gfCNCPoint3[16834] = {X 95.6267, Y 61.5566, Z -4.6667, A 0.000, B 0.000, C 0.000 }
gfCNCPoint3[16835] = {X 93.9906, Y 61.7990, Z -4.6667, A 0.000, B 0.000, C 0.000 }
gfCNCPoint3[16836] = {X 92.3385, Y 61.8800, Z -4.6667, A 0.000, B 0.000, C 0.000 }
gfCNCPoint3[16837] = {X 85.8951, Y 61.8800, Z -4.6667, A 0.000, B 0.000, C 0.000 }
gfCNCPoint3[16838] = {X 85.1609, Y 61.8640, Z -4.6667, A 0.000, B 0.000, C 0.000 }
gfCNCPoint3[16839] = {X 84.4280, Y 61.8161, Z -4.6667, A 0.000, B 0.000, C 0.000 }
gfCNCPoint3[16840] = {X 82.7247, Y 63.0692, Z -4.6667, A 0.000, B 0.000, C 0.000 }
gfCNCPoint3[16841] = {X 80.9073, Y 64.1504, Z -4.6667, A 0.000, B 0.000, C 0.000 }
gfCNCPoint3[16842] = {X 78.9932, Y 65.0494, Z -4.6667, A 0.000, B 0.000, C 0.000 }
gfCNCPoint3[16843] = {X 77.0007, Y 65.7577, Z -4.6667, A 0.000, B 0.000, C 0.000 }
gfCNCPoint3[16844] = {X 74.9487, Y 66.2685, Z -4.6667, A 0.000, B 0.000, C 0.000 }
gfCNCPoint3[16845] = {X 72.8566, Y 66.5769, Z -4.6667, A 0.000, B 0.000, C 0.000 }
gfCNCPoint3[16846] = {X 70.7445, Y 66.6800, Z -4.6667, A 0.000, B 0.000, C 0.000 }
gfCNCPoint3[16847] = {X 64.1851, Y 66.6800, Z -4.6667, A 0.000, B 0.000, C 0.000 }
gfCNCPoint3[16848] = {X 62.0576, Y 66.5754, Z -4.6667, A 0.000, B 0.000, C 0.000 }
gfCNCPoint3[16849] = {X 59.9505, Y 66.2624, Z -4.6667, A 0.000, B 0.000, C 0.000 }
gfCNCPoint3[16850] = {X 57.8844, Y 65.7442, Z -4.6667, A 0.000, B 0.000, C 0.000 }
gfCNCPoint3[16851] = {X 55.8790, Y 65.0258, Z -4.6667, A 0.000, B 0.000, C 0.000 }
gfCNCPoint3[16852] = {X 53.8737, Y 65.7442, Z -4.6667, A 0.000, B 0.000, C 0.000 }
gfCNCPoint3[16853] = {X 51.8075, Y 66.2624, Z -4.6667, A 0.000, B 0.000, C 0.000 }
gfCNCPoint3[16854] = {X 49.7005, Y 66.5754, Z -4.6667, A 0.000, B 0.000, C 0.000 }
gfCNCPoint3[16855] = {X 47.5729, Y 66.6800, Z -4.6667, A 0.000, B 0.000, C 0.000 }
gfCNCPoint3[16856] = {X 40.6393, Y 66.6800, Z -4.6667, A 0.000, B 0.000, C 0.000 }
gfCNCPoint3[16857] = {X 38.5447, Y 66.5786, Z -4.6667, A 0.000, B 0.000, C 0.000 }
gfCNCPoint3[16858] = {X 36.4697, Y 66.2753, Z -4.6667, A 0.000, B 0.000, C 0.000 }
gfCNCPoint3[16859] = {X 34.5048, Y 67.0013, Z -4.6667, A 0.000, B 0.000, C 0.000 }
gfCNCPoint3[16860] = {X 32.4879, Y 67.5668, Z -4.6667, A 0.000, B 0.000, C 0.000 }
gfCNCPoint3[16861] = {X 30.4319, Y 67.9682, Z -4.6667, A 0.000, B 0.000, C 0.000 }
gfCNCPoint3[16862] = {X 28.4180, Y 68.7658, Z -4.6667, A 0.000, B 0.000, C 0.000 }
gfCNCPoint3[16863] = {X 26.3720, Y 69.4768, Z -4.6667, A 0.000, B 0.000, C 0.000 }
gfCNCPoint3[16864] = {X 23.9561, Y 70.1952, Z -4.6667, A 0.000, B 0.000, C 0.000 }
gfCNCPoint3[16865] = {X 21.5034, Y 70.7756, Z -4.6667, A 0.000, B 0.000, C 0.000 }
gfCNCPoint3[16866] = {X 21.5034, Y 78.4950, Z -4.6667, A 0.000, B 0.000, C 0.000 }
gfCNCPoint3[16867] = {X 109.6713, Y 78.4950, Z -4.6667, A 0.000, B 0.000, C 0.000 }
gfCNCPoint3[16868] = {X 111.3427, Y 77.2335, Z -4.6667, A 0.000, B 0.000, C 0.000 }
gfCNCPoint3[16869] = {X 113.1173, Y 76.1220, Z -4.6667, A 0.000, B 0.000, C 0.000 }
gfCNCPoint3[16870] = {X 114.9818, Y 75.1689, Z -4.6667, A 0.000, B 0.000, C 0.000 }
gfCNCPoint3[16871] = {X 116.9220, Y 74.3813, Z -4.6667, A 0.000, B 0.000, C 0.000 }
gfCNCPoint3[16872] = {X 130.4111, Y 59.5684, Z -4.6667, A 0.000, B 0.000, C 0.000 }
gfCNCPoint3[16873] = {X 129.5278, Y 58.7531, Z -4.6667, A 0.000, B 0.000, C 0.000 }
gfCNCPoint3[16874] = {X 128.6970, Y 57.8844, Z -4.6667, A 0.000, B 0.000, C 0.000 }
gfCNCPoint3[16875] = {X 127.3929, Y 58.8834, Z -4.6667, A 0.000, B 0.000, C 0.000 }
gfCNCPoint3[16876] = {X 125.9978, Y 59.7510, Z -4.6667, A 0.000, B 0.000, C 0.000 }
gfCNCPoint3[16877] = {X 124.5250, Y 60.4789, Z -4.6667, A 0.000, B 0.000, C 0.000 }
gfCNCPoint3[16878] = {X 122.9885, Y 61.0601, Z -4.6667, A 0.000, B 0.000, C 0.000 }
gfCNCPoint3[16879] = {X 121.2879, Y 61.5139, Z -4.6667, A 0.000, B 0.000, C 0.000 }
gfCNCPoint3[16880] = {X 119.5493, Y 61.7882, Z -4.6667, A 0.000, B 0.000, C 0.000 }
gfCNCPoint3[16881] = {X 117.7916, Y 61.8800, Z -4.6667, A 0.000, B 0.000, C 0.000 }
gfCNCPoint3[16882] = {X 111.9185, Y 61.8800, Z -4.6667, A 0.000, B 0.000, C 0.000 }
gfCNCPoint3[16883] = {X 111.6170, Y 61.8773, Z -4.6667, A 0.000, B 0.000, C 0.000 }
gfCNCPoint3[16884] = {X 111.3156, Y 61.8692, Z -4.6667, A 0.000, B 0.000, C 0.000 }
gfCNCPoint3[16885] = {X 111.4013, Y 59.4708, Z -4.6667, A 0.000, B 0.000, C 0.000 }
gfCNCPoint3[16886] = {X 109.9149, Y 59.3407, Z -4.6667, A 0.000, B 0.000, C 0.000 }
gfCNCPoint3[16887] = {X 108.4496, Y 59.0584, Z -4.6667, A 0.000, B 0.000, C 0.000 }
gfCNCPoint3[16888] = {X 107.0213, Y 58.6267, Z -4.6667, A 0.000, B 0.000, C 0.000 }
gfCNCPoint3[16889] = {X 105.4260, Y 59.0985, Z -4.6667, A 0.000, B 0.000, C 0.000 }
gfCNCPoint3[16890] = {X 103.7872, Y 59.3842, Z -4.6667, A 0.000, B 0.000, C 0.000 }
gfCNCPoint3[16891] = {X 102.1264, Y 59.4800, Z -4.6667, A 0.000, B 0.000, C 0.000 }
gfCNCPoint3[16892] = {X 100.4656, Y 59.3847, Z -4.6667, A 0.000, B 0.000, C 0.000 }
gfCNCPoint3[16893] = {X 98.8267, Y 59.0996, Z -4.6667, A 0.000, B 0.000, C 0.000 }
gfCNCPoint3[16894] = {X 97.2313, Y 58.6283, Z -4.6667, A 0.000, B 0.000, C 0.000 }
gfCNCPoint3[16895] = {X 95.6367, Y 59.0994, Z -4.6667, A 0.000, B 0.000, C 0.000 }
gfCNCPoint3[16896] = {X 93.9986, Y 59.3845, Z -4.6667, A 0.000, B 0.000, C 0.000 }
gfCNCPoint3[16897] = {X 92.3385, Y 59.4800, Z -4.6667, A 0.000, B 0.000, C 0.000 }
gfCNCPoint3[16898] = {X 85.8951, Y 59.4800, Z -4.6667, A 0.000, B 0.000, C 0.000 }
gfCNCPoint3[16899] = {X 84.7780, Y 59.4368, Z -4.6667, A 0.000, B 0.000, C 0.000 }
gfCNCPoint3[16900] = {X 83.6677, Y 59.3077, Z -4.6667, A 0.000, B 0.000, C 0.000 }
gfCNCPoint3[16901] = {X 82.0978, Y 60.5827, Z -4.6667, A 0.000, B 0.000, C 0.000 }
gfCNCPoint3[16902] = {X 80.4031, Y 61.6862, Z -4.6667, A 0.000, B 0.000, C 0.000 }
gfCNCPoint3[16903] = {X 78.6021, Y 62.6061, Z -4.6667, A 0.000, B 0.000, C 0.000 }
gfCNCPoint3[16904] = {X 76.7146, Y 63.3324, Z -4.6667, A 0.000, B 0.000, C 0.000 }
gfCNCPoint3[16905] = {X 74.7614, Y 63.8569, Z -4.6667, A 0.000, B 0.000, C 0.000 }
gfCNCPoint3[16906] = {X 72.7640, Y 64.1739, Z -4.6667, A 0.000, B 0.000, C 0.000 }
gfCNCPoint3[16907] = {X 70.7445, Y 64.2800, Z -4.6667, A 0.000, B 0.000, C 0.000 }
gfCNCPoint3[16908] = {X 64.1851, Y 64.2800, Z -4.6667, A 0.000, B 0.000, C 0.000 }
gfCNCPoint3[16909] = {X 62.0428, Y 64.1606, Z -4.6667, A 0.000, B 0.000, C 0.000 }
gfCNCPoint3[16910] = {X 59.9269, Y 63.8039, Z -4.6667, A 0.000, B 0.000, C 0.000 }
gfCNCPoint3[16911] = {X 57.8638, Y 63.2143, Z -4.6667, A 0.000, B 0.000, C 0.000 }
gfCNCPoint3[16912] = {X 55.8790, Y 62.3991, Z -4.6667, A 0.000, B 0.000, C 0.000 }
gfCNCPoint3[16913] = {X 53.8942, Y 63.2143, Z -4.6667, A 0.000, B 0.000, C 0.000 }
gfCNCPoint3[16914] = {X 51.8311, Y 63.8039, Z -4.6667, A 0.000, B 0.000, C 0.000 }
gfCNCPoint3[16915] = {X 49.7153, Y 64.1606, Z -4.6667, A 0.000, B 0.000, C 0.000 }
gfCNCPoint3[16916] = {X 47.5729, Y 64.2800, Z -4.6667, A 0.000, B 0.000, C 0.000 }
gfCNCPoint3[16917] = {X 40.6393, Y 64.2800, Z -4.6667, A 0.000, B 0.000, C 0.000 }
gfCNCPoint3[16918] = {X 39.1549, Y 64.2228, Z -4.6667, A 0.000, B 0.000, C 0.000 }
gfCNCPoint3[16919] = {X 37.6792, Y 64.0514, Z -4.6667, A 0.000, B 0.000, C 0.000 }
gfCNCPoint3[16920] = {X 36.2212, Y 63.7670, Z -4.6667, A 0.000, B 0.000, C 0.000 }
gfCNCPoint3[16921] = {X 34.1358, Y 64.5944, Z -4.6667, A 0.000, B 0.000, C 0.000 }
gfCNCPoint3[16922] = {X 31.9814, Y 65.2203, Z -4.6667, A 0.000, B 0.000, C 0.000 }
gfCNCPoint3[16923] = {X 29.7773, Y 65.6388, Z -4.6667, A 0.000, B 0.000, C 0.000 }
gfCNCPoint3[16924] = {X 27.7204, Y 66.4644, Z -4.6667, A 0.000, B 0.000, C 0.000 }
gfCNCPoint3[16925] = {X 25.6278, Y 67.1951, Z -4.6667, A 0.000, B 0.000, C 0.000 }
gfCNCPoint3[16926] = {X 23.4821, Y 67.8375, Z -4.6667, A 0.000, B 0.000, C 0.000 }
gfCNCPoint3[16927] = {X 21.3053, Y 68.3647, Z -4.6667, A 0.000, B 0.000, C 0.000 }
gfCNCPoint3[16928] = {X 19.1034, Y 68.7753, Z -4.6667, A 0.000, B 0.000, C 0.000 }
gfCNCPoint3[16929] = {X 19.1034, Y 80.8950, Z -4.6667, A 0.000, B 0.000, C 0.000 }
gfCNCPoint3[16930] = {X 110.5596, Y 80.8950, Z -4.6667, A 0.000, B 0.000, C 0.000 }
gfCNCPoint3[16931] = {X 112.3069, Y 79.4902, Z -4.6667, A 0.000, B 0.000, C 0.000 }
gfCNCPoint3[16932] = {X 114.1898, Y 78.2733, Z -4.6667, A 0.000, B 0.000, C 0.000 }
gfCNCPoint3[16933] = {X 116.1884, Y 77.2574, Z -4.6667, A 0.000, B 0.000, C 0.000 }
gfCNCPoint3[16934] = {X 118.2812, Y 76.4533, Z -4.6667, A 0.000, B 0.000, C 0.000 }
gfCNCPoint3[16935] = {X 133.9633, Y 59.2322, Z -4.6667, A 0.000, B 0.000, C 0.000 }
gfCNCPoint3[16936] = {X 132.7155, Y 58.3546, Z -4.6667, A 0.000, B 0.000, C 0.000 }
gfCNCPoint3[16937] = {X 131.5520, Y 57.3681, Z -4.6667, A 0.000, B 0.000, C 0.000 }
gfCNCPoint3[16938] = {X 130.4824, Y 56.2805, Z -4.6667, A 0.000, B 0.000, C 0.000 }
gfCNCPoint3[16939] = {X 129.6655, Y 55.2988, Z -4.6667, A 0.000, B 0.000, C 0.000 }
gfCNCPoint3[16940] = {X 128.9251, Y 54.2582, Z -4.6667, A 0.000, B 0.000, C 0.000 }
gfCNCPoint3[16941] = {X 128.0750, Y 55.1942, Z -4.6667, A 0.000, B 0.000, C 0.000 }
gfCNCPoint3[16942] = {X 127.1464, Y 56.0525, Z -4.6667, A 0.000, B 0.000, C 0.000 }
gfCNCPoint3[16943] = {X 125.7915, Y 57.0695, Z -4.6667, A 0.000, B 0.000, C 0.000 }
gfCNCPoint3[16944] = {X 124.3270, Y 57.9212, Z -4.6667, A 0.000, B 0.000, C 0.000 }
gfCNCPoint3[16945] = {X 122.7731, Y 58.5961, Z -4.6667, A 0.000, B 0.000, C 0.000 }
gfCNCPoint3[16946] = {X 121.1510, Y 59.0849, Z -4.6667, A 0.000, B 0.000, C 0.000 }
gfCNCPoint3[16947] = {X 119.4828, Y 59.3809, Z -4.6667, A 0.000, B 0.000, C 0.000 }
gfCNCPoint3[16948] = {X 117.7916, Y 59.4800, Z -4.6667, A 0.000, B 0.000, C 0.000 }
gfCNCPoint3[16949] = {X 111.9185, Y 59.4800, Z -4.6667, A 0.000, B 0.000, C 0.000 }
gfCNCPoint3[16950] = {X 111.6599, Y 59.4777, Z -4.6667, A 0.000, B 0.000, C 0.000 }
gfCNCPoint3[16951] = {X 111.4013, Y 59.4708, Z -4.6667, A 0.000, B 0.000, C 0.000 }
gfCNCPoint3[16952] = {X 111.4871, Y 57.0723, Z -4.6667, A 0.000, B 0.000, C 0.000 }
gfCNCPoint3[16953] = {X 109.9587, Y 56.9200, Z -4.6667, A 0.000, B 0.000, C 0.000 }
gfCNCPoint3[16954] = {X 108.4621, Y 56.5750, Z -4.6667, A 0.000, B 0.000, C 0.000 }
gfCNCPoint3[16955] = {X 107.0213, Y 56.0428, Z -4.6667, A 0.000, B 0.000, C 0.000 }
gfCNCPoint3[16956] = {X 105.4432, Y 56.6151, Z -4.6667, A 0.000, B 0.000, C 0.000 }
gfCNCPoint3[16957] = {X 103.8010, Y 56.9630, Z -4.6667, A 0.000, B 0.000, C 0.000 }
gfCNCPoint3[16958] = {X 102.1265, Y 57.0800, Z -4.6667, A 0.000, B 0.000, C 0.000 }
gfCNCPoint3[16959] = {X 100.4519, Y 56.9637, Z -4.6667, A 0.000, B 0.000, C 0.000 }
gfCNCPoint3[16960] = {X 98.8096, Y 56.6164, Z -4.6667, A 0.000, B 0.000, C 0.000 }
gfCNCPoint3[16961] = {X 97.2313, Y 56.0448, Z -4.6667, A 0.000, B 0.000, C 0.000 }
gfCNCPoint3[16962] = {X 95.6538, Y 56.6162, Z -4.6667, A 0.000, B 0.000, C 0.000 }
gfCNCPoint3[16963] = {X 94.0123, Y 56.9635, Z -4.6667, A 0.000, B 0.000, C 0.000 }
gfCNCPoint3[16964] = {X 92.3385, Y 57.0800, Z -4.6667, A 0.000, B 0.000, C 0.000 }
gfCNCPoint3[16965] = {X 85.8951, Y 57.0800, Z -4.6667, A 0.000, B 0.000, C 0.000 }
gfCNCPoint3[16966] = {X 84.3894, Y 56.9858, Z -4.6667, A 0.000, B 0.000, C 0.000 }
gfCNCPoint3[16967] = {X 82.9073, Y 56.7047, Z -4.6667, A 0.000, B 0.000, C 0.000 }
gfCNCPoint3[16968] = {X 81.4847, Y 58.0224, Z -4.6667, A 0.000, B 0.000, C 0.000 }
gfCNCPoint3[16969] = {X 79.9203, Y 59.1682, Z -4.6667, A 0.000, B 0.000, C 0.000 }
gfCNCPoint3[16970] = {X 78.2348, Y 60.1271, Z -4.6667, A 0.000, B 0.000, C 0.000 }
gfCNCPoint3[16971] = {X 76.4504, Y 60.8864, Z -4.6667, A 0.000, B 0.000, C 0.000 }
gfCNCPoint3[16972] = {X 74.5908, Y 61.4359, Z -4.6667, A 0.000, B 0.000, C 0.000 }
gfCNCPoint3[16973] = {X 72.6804, Y 61.7686, Z -4.6667, A 0.000, B 0.000, C 0.000 }
gfCNCPoint3[16974] = {X 70.7445, Y 61.8800, Z -4.6667, A 0.000, B 0.000, C 0.000 }
gfCNCPoint3[16975] = {X 64.1851, Y 61.8800, Z -4.6667, A 0.000, B 0.000, C 0.000 }
gfCNCPoint3[16976] = {X 62.4514, Y 61.7907, Z -4.6667, A 0.000, B 0.000, C 0.000 }
gfCNCPoint3[16977] = {X 60.7359, Y 61.5238, Z -4.6667, A 0.000, B 0.000, C 0.000 }
gfCNCPoint3[16978] = {X 59.0570, Y 61.0822, Z -4.6667, A 0.000, B 0.000, C 0.000 }
gfCNCPoint3[16979] = {X 57.4323, Y 60.4704, Z -4.6667, A 0.000, B 0.000, C 0.000 }
gfCNCPoint3[16980] = {X 55.8790, Y 59.6950, Z -4.6667, A 0.000, B 0.000, C 0.000 }
gfCNCPoint3[16981] = {X 54.3258, Y 60.4704, Z -4.6667, A 0.000, B 0.000, C 0.000 }
gfCNCPoint3[16982] = {X 52.7011, Y 61.0822, Z -4.6667, A 0.000, B 0.000, C 0.000 }
gfCNCPoint3[16983] = {X 51.0221, Y 61.5238, Z -4.6667, A 0.000, B 0.000, C 0.000 }
gfCNCPoint3[16984] = {X 49.3067, Y 61.7907, Z -4.6667, A 0.000, B 0.000, C 0.000 }
gfCNCPoint3[16985] = {X 47.5729, Y 61.8800, Z -4.6667, A 0.000, B 0.000, C 0.000 }
gfCNCPoint3[16986] = {X 40.6393, Y 61.8800, Z -4.6667, A 0.000, B 0.000, C 0.000 }
gfCNCPoint3[16987] = {X 39.0678, Y 61.8067, Z -4.6667, A 0.000, B 0.000, C 0.000 }
gfCNCPoint3[16988] = {X 37.5100, Y 61.5874, Z -4.6667, A 0.000, B 0.000, C 0.000 }
gfCNCPoint3[16989] = {X 35.9793, Y 61.2240, Z -4.6667, A 0.000, B 0.000, C 0.000 }
gfCNCPoint3[16990] = {X 34.3394, Y 61.9603, Z -4.6667, A 0.000, B 0.000, C 0.000 }
gfCNCPoint3[16991] = {X 32.6430, Y 62.5550, Z -4.6667, A 0.000, B 0.000, C 0.000 }
gfCNCPoint3[16992] = {X 30.9023, Y 63.0040, Z -4.6667, A 0.000, B 0.000, C 0.000 }
gfCNCPoint3[16993] = {X 29.1299, Y 63.3040, Z -4.6667, A 0.000, B 0.000, C 0.000 }
gfCNCPoint3[16994] = {X 27.0266, Y 64.1611, Z -4.6667, A 0.000, B 0.000, C 0.000 }
gfCNCPoint3[16995] = {X 24.8836, Y 64.9134, Z -4.6667, A 0.000, B 0.000, C 0.000 }
gfCNCPoint3[16996] = {X 22.2005, Y 65.6920, Z -4.6667, A 0.000, B 0.000, C 0.000 }
gfCNCPoint3[16997] = {X 19.4693, Y 66.2797, Z -4.6667, A 0.000, B 0.000, C 0.000 }
gfCNCPoint3[16998] = {X 16.7034, Y 66.6737, Z -4.6667, A 0.000, B 0.000, C 0.000 }
gfCNCPoint3[16999] = {X 16.7034, Y 83.2950, Z -4.6667, A 0.000, B 0.000, C 0.000 }
gfCNCPoint3[17000] = {X 111.5063, Y 83.2950, Z -4.6667, A 0.000, B 0.000, C 0.000 }
gfCNCPoint3[17001] = {X 112.9249, Y 82.0356, Z -4.6667, A 0.000, B 0.000, C 0.000 }
gfCNCPoint3[17002] = {X 114.4604, Y 80.9217, Z -4.6667, A 0.000, B 0.000, C 0.000 }
gfCNCPoint3[17003] = {X 116.0979, Y 79.9641, Z -4.6667, A 0.000, B 0.000, C 0.000 }
gfCNCPoint3[17004] = {X 117.8217, Y 79.1721, Z -4.6667, A 0.000, B 0.000, C 0.000 }
gfCNCPoint3[17005] = {X 119.6149, Y 78.5533, Z -4.6667, A 0.000, B 0.000, C 0.000 }
gfCNCPoint3[17006] = {X 137.8571, Y 58.5208, Z -4.6667, A 0.000, B 0.000, C 0.000 }
gfCNCPoint3[17007] = {X 136.5223, Y 57.9304, Z -4.6667, A 0.000, B 0.000, C 0.000 }
gfCNCPoint3[17008] = {X 135.2537, Y 57.2086, Z -4.6667, A 0.000, B 0.000, C 0.000 }
gfCNCPoint3[17009] = {X 134.0098, Y 56.3196, Z -4.6667, A 0.000, B 0.000, C 0.000 }
gfCNCPoint3[17010] = {X 132.8666, Y 55.3044, Z -4.6667, A 0.000, B 0.000, C 0.000 }
gfCNCPoint3[17011] = {X 131.8368, Y 54.1743, Z -4.6667, A 0.000, B 0.000, C 0.000 }
gfCNCPoint3[17012] = {X 130.9319, Y 52.9419, Z -4.6667, A 0.000, B 0.000, C 0.000 }
gfCNCPoint3[17013] = {X 130.2147, Y 51.7225, Z -4.6667, A 0.000, B 0.000, C 0.000 }
gfCNCPoint3[17014] = {X 129.6199, Y 50.4390, Z -4.6667, A 0.000, B 0.000, C 0.000 }
gfCNCPoint3[17015] = {X 129.1532, Y 49.1035, Z -4.6667, A 0.000, B 0.000, C 0.000 }
gfCNCPoint3[17016] = {X 128.6036, Y 50.3877, Z -4.6667, A 0.000, B 0.000, C 0.000 }
gfCNCPoint3[17017] = {X 127.9093, Y 51.5998, Z -4.6667, A 0.000, B 0.000, C 0.000 }
gfCNCPoint3[17018] = {X 127.0798, Y 52.7237, Z -4.6667, A 0.000, B 0.000, C 0.000 }
gfCNCPoint3[17019] = {X 126.0417, Y 53.8239, Z -4.6667, A 0.000, B 0.000, C 0.000 }
gfCNCPoint3[17020] = {X 124.8743, Y 54.7858, Z -4.6667, A 0.000, B 0.000, C 0.000 }
gfCNCPoint3[17021] = {X 123.5958, Y 55.5942, Z -4.6667, A 0.000, B 0.000, C 0.000 }
gfCNCPoint3[17022] = {X 122.2263, Y 56.2365, Z -4.6667, A 0.000, B 0.000, C 0.000 }
gfCNCPoint3[17023] = {X 120.7872, Y 56.7027, Z -4.6667, A 0.000, B 0.000, C 0.000 }
gfCNCPoint3[17024] = {X 119.3012, Y 56.9853, Z -4.6667, A 0.000, B 0.000, C 0.000 }
gfCNCPoint3[17025] = {X 117.7916, Y 57.0800, Z -4.6667, A 0.000, B 0.000, C 0.000 }
gfCNCPoint3[17026] = {X 111.9185, Y 57.0800, Z -4.6667, A 0.000, B 0.000, C 0.000 }
gfCNCPoint3[17027] = {X 111.7027, Y 57.0781, Z -4.6667, A 0.000, B 0.000, C 0.000 }
gfCNCPoint3[17028] = {X 111.4871, Y 57.0723, Z -4.6667, A 0.000, B 0.000, C 0.000 }
gfCNCPoint3[17029] = {X 111.5728, Y 54.6738, Z -4.6667, A 0.000, B 0.000, C 0.000 }
gfCNCPoint3[17030] = {X 110.3820, Y 54.5573, Z -4.6667, A 0.000, B 0.000, C 0.000 }
gfCNCPoint3[17031] = {X 109.2147, Y 54.2947, Z -4.6667, A 0.000, B 0.000, C 0.000 }
gfCNCPoint3[17032] = {X 108.0887, Y 53.8902, Z -4.6667, A 0.000, B 0.000, C 0.000 }
gfCNCPoint3[17033] = {X 107.0213, Y 53.3498, Z -4.6667, A 0.000, B 0.000, C 0.000 }
gfCNCPoint3[17034] = {X 106.6480, Y 53.5578, Z -4.6667, A 0.000, B 0.000, C 0.000 }
gfCNCPoint3[17035] = {X 106.2658, Y 53.7492, Z -4.6667, A 0.000, B 0.000, C 0.000 }
gfCNCPoint3[17036] = {X 105.0149, Y 54.2383, Z -4.6667, A 0.000, B 0.000, C 0.000 }
gfCNCPoint3[17037] = {X 103.7084, Y 54.5495, Z -4.6667, A 0.000, B 0.000, C 0.000 }
gfCNCPoint3[17038] = {X 102.3713, Y 54.6768, Z -4.6667, A 0.000, B 0.000, C 0.000 }
gfCNCPoint3[17039] = {X 101.0295, Y 54.6179, Z -4.6667, A 0.000, B 0.000, C 0.000 }
gfCNCPoint3[17040] = {X 99.7088, Y 54.3738, Z -4.6667, A 0.000, B 0.000, C 0.000 }
gfCNCPoint3[17041] = {X 98.4345, Y 53.9493, Z -4.6667, A 0.000, B 0.000, C 0.000 }
gfCNCPoint3[17042] = {X 97.2313, Y 53.3524, Z -4.6667, A 0.000, B 0.000, C 0.000 }
gfCNCPoint3[17043] = {X 96.0852, Y 53.9255, Z -4.6667, A 0.000, B 0.000, C 0.000 }
gfCNCPoint3[17044] = {X 94.8734, Y 54.3422, Z -4.6667, A 0.000, B 0.000, C 0.000 }
gfCNCPoint3[17045] = {X 93.6172, Y 54.5952, Z -4.6667, A 0.000, B 0.000, C 0.000 }
gfCNCPoint3[17046] = {X 92.3385, Y 54.6800, Z -4.6667, A 0.000, B 0.000, C 0.000 }
gfCNCPoint3[17047] = {X 85.8951, Y 54.6800, Z -4.6667, A 0.000, B 0.000, C 0.000 }
gfCNCPoint3[17048] = {X 84.6159, Y 54.5951, Z -4.6667, A 0.000, B 0.000, C 0.000 }
gfCNCPoint3[17049] = {X 83.3592, Y 54.3419, Z -4.6667, A 0.000, B 0.000, C 0.000 }
gfCNCPoint3[17050] = {X 82.1469, Y 53.9249, Z -4.6667, A 0.000, B 0.000, C 0.000 }
gfCNCPoint3[17051] = {X 81.0644, Y 55.1572, Z -4.6667, A 0.000, B 0.000, C 0.000 }
gfCNCPoint3[17052] = {X 79.8495, Y 56.2591, Z -4.6667, A 0.000, B 0.000, C 0.000 }
gfCNCPoint3[17053] = {X 78.5178, Y 57.2166, Z -4.6667, A 0.000, B 0.000, C 0.000 }
gfCNCPoint3[17054] = {X 77.0863, Y 58.0174, Z -4.6667, A 0.000, B 0.000, C 0.000 }
gfCNCPoint3[17055] = {X 75.5734, Y 58.6511, Z -4.6667, A 0.000, B 0.000, C 0.000 }
gfCNCPoint3[17056] = {X 73.9986, Y 59.1096, Z -4.6667, A 0.000, B 0.000, C 0.000 }
gfCNCPoint3[17057] = {X 72.3820, Y 59.3871, Z -4.6667, A 0.000, B 0.000, C 0.000 }
gfCNCPoint3[17058] = {X 70.7445, Y 59.4800, Z -4.6667, A 0.000, B 0.000, C 0.000 }
gfCNCPoint3[17059] = {X 64.1851, Y 59.4800, Z -4.6667, A 0.000, B 0.000, C 0.000 }
gfCNCPoint3[17060] = {X 62.4203, Y 59.3720, Z -4.6667, A 0.000, B 0.000, C 0.000 }
gfCNCPoint3[17061] = {X 60.6818, Y 59.0498, Z -4.6667, A 0.000, B 0.000, C 0.000 }
gfCNCPoint3[17062] = {X 58.9955, Y 58.5181, Z -4.6667, A 0.000, B 0.000, C 0.000 }
gfCNCPoint3[17063] = {X 57.3866, Y 57.7848, Z -4.6667, A 0.000, B 0.000, C 0.000 }
gfCNCPoint3[17064] = {X 55.8790, Y 56.8608, Z -4.6667, A 0.000, B 0.000, C 0.000 }
gfCNCPoint3[17065] = {X 54.3715, Y 57.7848, Z -4.6667, A 0.000, B 0.000, C 0.000 }
gfCNCPoint3[17066] = {X 52.7626, Y 58.5181, Z -4.6667, A 0.000, B 0.000, C 0.000 }
gfCNCPoint3[17067] = {X 51.0763, Y 59.0498, Z -4.6667, A 0.000, B 0.000, C 0.000 }
gfCNCPoint3[17068] = {X 49.3378, Y 59.3720, Z -4.6667, A 0.000, B 0.000, C 0.000 }
gfCNCPoint3[17069] = {X 47.5729, Y 59.4800, Z -4.6667, A 0.000, B 0.000, C 0.000 }
gfCNCPoint3[17070] = {X 40.6393, Y 59.4800, Z -4.6667, A 0.000, B 0.000, C 0.000 }
gfCNCPoint3[17071] = {X 38.9797, Y 59.3846, Z -4.6667, A 0.000, B 0.000, C 0.000 }
gfCNCPoint3[17072] = {X 37.3419, Y 59.0996, Z -4.6667, A 0.000, B 0.000, C 0.000 }
gfCNCPoint3[17073] = {X 35.7476, Y 58.6287, Z -4.6667, A 0.000, B 0.000, C 0.000 }
gfCNCPoint3[17074] = {X 34.0326, Y 59.4873, Z -4.6667, A 0.000, B 0.000, C 0.000 }
gfCNCPoint3[17075] = {X 32.2391, Y 60.1668, Z -4.6667, A 0.000, B 0.000, C 0.000 }
gfCNCPoint3[17076] = {X 30.3858, Y 60.6602, Z -4.6667, A 0.000, B 0.000, C 0.000 }
gfCNCPoint3[17077] = {X 28.4918, Y 60.9624, Z -4.6667, A 0.000, B 0.000, C 0.000 }
gfCNCPoint3[17078] = {X 26.3379, Y 61.8552, Z -4.6667, A 0.000, B 0.000, C 0.000 }
gfCNCPoint3[17079] = {X 24.1393, Y 62.6318, Z -4.6667, A 0.000, B 0.000, C 0.000 }
gfCNCPoint3[17080] = {X 21.7320, Y 63.3348, Z -4.6667, A 0.000, B 0.000, C 0.000 }
gfCNCPoint3[17081] = {X 19.2828, Y 63.8743, Z -4.6667, A 0.000, B 0.000, C 0.000 }
gfCNCPoint3[17082] = {X 16.8029, Y 64.2478, Z -4.6667, A 0.000, B 0.000, C 0.000 }
gfCNCPoint3[17083] = {X 14.3034, Y 64.4536, Z -4.6667, A 0.000, B 0.000, C 0.000 }
gfCNCPoint3[17084] = {X 14.3034, Y 85.6950, Z -4.6667, A 0.000, B 0.000, C 0.000 }
gfCNCPoint3[17085] = {X 112.5245, Y 85.6950, Z -4.6667, A 0.000, B 0.000, C 0.000 }
gfCNCPoint3[17086] = {X 113.9434, Y 84.3111, Z -4.6667, A 0.000, B 0.000, C 0.000 }
gfCNCPoint3[17087] = {X 115.5147, Y 83.1030, Z -4.6667, A 0.000, B 0.000, C 0.000 }
gfCNCPoint3[17088] = {X 117.2168, Y 82.0874, Z -4.6667, A 0.000, B 0.000, C 0.000 }
gfCNCPoint3[17089] = {X 119.0261, Y 81.2784, Z -4.6667, A 0.000, B 0.000, C 0.000 }
gfCNCPoint3[17090] = {X 120.9179, Y 80.6870, Z -4.6667, A 0.000, B 0.000, C 0.000 }
gfCNCPoint3[17091] = {X 142.4291, Y 57.0646, Z -4.6667, A 0.000, B 0.000, C 0.000 }
gfCNCPoint3[17092] = {X 141.1662, Y 56.9338, Z -4.6667, A 0.000, B 0.000, C 0.000 }
gfCNCPoint3[17093] = {X 139.9239, Y 56.6713, Z -4.6667, A 0.000, B 0.000, C 0.000 }
gfCNCPoint3[17094] = {X 138.7160, Y 56.2798, Z -4.6667, A 0.000, B 0.000, C 0.000 }
gfCNCPoint3[17095] = {X 137.2790, Y 55.6180, Z -4.6667, A 0.000, B 0.000, C 0.000 }
gfCNCPoint3[17096] = {X 135.9408, Y 54.7741, Z -4.6667, A 0.000, B 0.000, C 0.000 }
gfCNCPoint3[17097] = {X 134.7243, Y 53.7625, Z -4.6667, A 0.000, B 0.000, C 0.000 }
gfCNCPoint3[17098] = {X 133.6505, Y 52.6007, Z -4.6667, A 0.000, B 0.000, C 0.000 }
gfCNCPoint3[17099] = {X 132.7377, Y 51.3084, Z -4.6667, A 0.000, B 0.000, C 0.000 }
gfCNCPoint3[17100] = {X 132.0016, Y 49.9080, Z -4.6667, A 0.000, B 0.000, C 0.000 }
gfCNCPoint3[17101] = {X 131.4549, Y 48.4234, Z -4.6667, A 0.000, B 0.000, C 0.000 }
gfCNCPoint3[17102] = {X 131.1845, Y 47.3200, Z -4.6667, A 0.000, B 0.000, C 0.000 }
gfCNCPoint3[17103] = {X 131.0190, Y 46.1961, Z -4.6667, A 0.000, B 0.000, C 0.000 }
gfCNCPoint3[17104] = {X 130.9598, Y 45.0616, Z -4.6667, A 0.000, B 0.000, C 0.000 }
gfCNCPoint3[17105] = {X 130.9601, Y 44.0978, Z -4.6667, A 0.000, B 0.000, C 0.000 }
gfCNCPoint3[17106] = {X 131.0921, Y 42.4244, Z -4.6667, A 0.000, B 0.000, C 0.000 }
gfCNCPoint3[17107] = {X 131.4548, Y 40.7854, Z -4.6667, A 0.000, B 0.000, C 0.000 }
gfCNCPoint3[17108] = {X 133.7565, Y 41.4655, Z -4.6667, A 0.000, B 0.000, C 0.000 }
gfCNCPoint3[17109] = {X 134.2330, Y 40.1906, Z -4.6667, A 0.000, B 0.000, C 0.000 }
gfCNCPoint3[17110] = {X 134.8836, Y 38.9952, Z -4.6667, A 0.000, B 0.000, C 0.000 }
gfCNCPoint3[17111] = {X 134.8836, Y 27.0854, Z -4.6667, A 0.000, B 0.000, C 0.000 }
gfCNCPoint3[17112] = {X 134.3931, Y 27.1259, Z -4.6667, A 0.000, B 0.000, C 0.000 }
gfCNCPoint3[17113] = {X 133.9011, Y 27.1414, Z -4.6667, A 0.000, B 0.000, C 0.000 }
gfCNCPoint3[17114] = {X 133.2006, Y 27.1415, Z -4.6667, A 0.000, B 0.000, C 0.000 }
gfCNCPoint3[17115] = {X 131.9567, Y 27.0613, Z -4.6667, A 0.000, B 0.000, C 0.000 }
gfCNCPoint3[17116] = {X 130.7333, Y 26.8218, Z -4.6667, A 0.000, B 0.000, C 0.000 }
gfCNCPoint3[17117] = {X 129.5509, Y 26.4271, Z -4.6667, A 0.000, B 0.000, C 0.000 }
gfCNCPoint3[17118] = {X 128.4290, Y 25.8838, Z -4.6667, A 0.000, B 0.000, C 0.000 }
gfCNCPoint3[17119] = {X 127.3862, Y 25.2007, Z -4.6667, A 0.000, B 0.000, C 0.000 }
gfCNCPoint3[17120] = {X 126.3456, Y 24.2961, Z -4.6667, A 0.000, B 0.000, C 0.000 }
gfCNCPoint3[17121] = {X 125.4440, Y 23.2527, Z -4.6667, A 0.000, B 0.000, C 0.000 }
gfCNCPoint3[17122] = {X 124.6999, Y 22.0918, Z -4.6667, A 0.000, B 0.000, C 0.000 }
gfCNCPoint3[17123] = {X 124.1282, Y 20.8370, Z -4.6667, A 0.000, B 0.000, C 0.000 }
gfCNCPoint3[17124] = {X 123.7407, Y 19.5136, Z -4.6667, A 0.000, B 0.000, C 0.000 }
gfCNCPoint3[17125] = {X 123.5451, Y 18.1486, Z -4.6667, A 0.000, B 0.000, C 0.000 }
gfCNCPoint3[17126] = {X 123.5441, Y 39.7471, Z -4.6667, A 0.000, B 0.000, C 0.000 }
gfCNCPoint3[17127] = {X 124.1926, Y 40.7410, Z -4.6667, A 0.000, B 0.000, C 0.000 }
gfCNCPoint3[17128] = {X 124.6710, Y 41.8272, Z -4.6667, A 0.000, B 0.000, C 0.000 }
gfCNCPoint3[17129] = {X 124.9665, Y 42.9766, Z -4.6667, A 0.000, B 0.000, C 0.000 }
gfCNCPoint3[17130] = {X 125.0714, Y 44.1587, Z -4.6667, A 0.000, B 0.000, C 0.000 }
gfCNCPoint3[17131] = {X 125.0716, Y 45.0000, Z -4.6667, A 0.000, B 0.000, C 0.000 }
gfCNCPoint3[17132] = {X 124.9610, Y 46.2642, Z -4.6667, A 0.000, B 0.000, C 0.000 }
gfCNCPoint3[17133] = {X 124.6325, Y 47.4899, Z -4.6667, A 0.000, B 0.000, C 0.000 }
gfCNCPoint3[17134] = {X 124.0962, Y 48.6400, Z -4.6667, A 0.000, B 0.000, C 0.000 }
gfCNCPoint3[17135] = {X 123.3684, Y 49.6795, Z -4.6667, A 0.000, B 0.000, C 0.000 }
gfCNCPoint3[17136] = {X 122.4711, Y 50.5768, Z -4.6667, A 0.000, B 0.000, C 0.000 }
gfCNCPoint3[17137] = {X 121.4316, Y 51.3047, Z -4.6667, A 0.000, B 0.000, C 0.000 }
gfCNCPoint3[17138] = {X 120.2815, Y 51.8410, Z -4.6667, A 0.000, B 0.000, C 0.000 }
gfCNCPoint3[17139] = {X 119.0557, Y 52.1694, Z -4.6667, A 0.000, B 0.000, C 0.000 }
gfCNCPoint3[17140] = {X 117.7916, Y 52.2800, Z -4.6667, A 0.000, B 0.000, C 0.000 }
gfCNCPoint3[17141] = {X 111.9185, Y 52.2800, Z -4.6667, A 0.000, B 0.000, C 0.000 }
gfCNCPoint3[17142] = {X 110.8481, Y 52.2009, Z -4.6667, A 0.000, B 0.000, C 0.000 }
gfCNCPoint3[17143] = {X 109.8009, Y 51.9652, Z -4.6667, A 0.000, B 0.000, C 0.000 }
gfCNCPoint3[17144] = {X 108.7998, Y 51.5782, Z -4.6667, A 0.000, B 0.000, C 0.000 }
gfCNCPoint3[17145] = {X 107.8665, Y 51.0481, Z -4.6667, A 0.000, B 0.000, C 0.000 }
gfCNCPoint3[17146] = {X 107.0213, Y 50.3866, Z -4.6667, A 0.000, B 0.000, C 0.000 }
gfCNCPoint3[17147] = {X 106.1743, Y 51.0493, Z -4.6667, A 0.000, B 0.000, C 0.000 }
gfCNCPoint3[17148] = {X 105.2389, Y 51.5800, Z -4.6667, A 0.000, B 0.000, C 0.000 }
gfCNCPoint3[17149] = {X 104.0917, Y 52.0091, Z -4.6667, A 0.000, B 0.000, C 0.000 }
gfCNCPoint3[17150] = {X 102.8887, Y 52.2397, Z -4.6667, A 0.000, B 0.000, C 0.000 }
gfCNCPoint3[17151] = {X 101.6641, Y 52.2655, Z -4.6667, A 0.000, B 0.000, C 0.000 }
gfCNCPoint3[17152] = {X 100.4526, Y 52.0855, Z -4.6667, A 0.000, B 0.000, C 0.000 }
gfCNCPoint3[17153] = {X 99.2883, Y 51.7050, Z -4.6667, A 0.000, B 0.000, C 0.000 }
gfCNCPoint3[17154] = {X 98.2043, Y 51.1347, Z -4.6667, A 0.000, B 0.000, C 0.000 }
gfCNCPoint3[17155] = {X 97.2313, Y 50.3907, Z -4.6667, A 0.000, B 0.000, C 0.000 }
gfCNCPoint3[17156] = {X 96.3865, Y 51.0508, Z -4.6667, A 0.000, B 0.000, C 0.000 }
gfCNCPoint3[17157] = {X 95.4539, Y 51.5797, Z -4.6667, A 0.000, B 0.000, C 0.000 }
gfCNCPoint3[17158] = {X 94.4538, Y 51.9659, Z -4.6667, A 0.000, B 0.000, C 0.000 }
gfCNCPoint3[17159] = {X 93.4078, Y 52.2011, Z -4.6667, A 0.000, B 0.000, C 0.000 }
gfCNCPoint3[17160] = {X 92.3385, Y 52.2800, Z -4.6667, A 0.000, B 0.000, C 0.000 }
gfCNCPoint3[17161] = {X 85.8951, Y 52.2800, Z -4.6667, A 0.000, B 0.000, C 0.000 }
gfCNCPoint3[17162] = {X 84.6852, Y 52.1788, Z -4.6667, A 0.000, B 0.000, C 0.000 }
gfCNCPoint3[17163] = {X 83.5090, Y 51.8779, Z -4.6667, A 0.000, B 0.000, C 0.000 }
gfCNCPoint3[17164] = {X 82.3992, Y 51.3857, Z -4.6667, A 0.000, B 0.000, C 0.000 }
gfCNCPoint3[17165] = {X 81.3866, Y 50.7159, Z -4.6667, A 0.000, B 0.000, C 0.000 }
gfCNCPoint3[17166] = {X 80.5223, Y 52.0937, Z -4.6667, A 0.000, B 0.000, C 0.000 }
gfCNCPoint3[17167] = {X 79.4808, Y 53.3429, Z -4.6667, A 0.000, B 0.000, C 0.000 }
gfCNCPoint3[17168] = {X 78.2809, Y 54.4408, Z -4.6667, A 0.000, B 0.000, C 0.000 }
gfCNCPoint3[17169] = {X 76.9444, Y 55.3676, Z -4.6667, A 0.000, B 0.000, C 0.000 }
gfCNCPoint3[17170] = {X 75.4955, Y 56.1065, Z -4.6667, A 0.000, B 0.000, C 0.000 }
gfCNCPoint3[17171] = {X 73.9605, Y 56.6440, Z -4.6667, A 0.000, B 0.000, C 0.000 }
gfCNCPoint3[17172] = {X 72.3672, Y 56.9705, Z -4.6667, A 0.000, B 0.000, C 0.000 }
gfCNCPoint3[17173] = {X 70.7445, Y 57.0800, Z -4.6667, A 0.000, B 0.000, C 0.000 }
gfCNCPoint3[17174] = {X 64.1851, Y 57.0800, Z -4.6667, A 0.000, B 0.000, C 0.000 }
gfCNCPoint3[17175] = {X 62.6628, Y 56.9837, Z -4.6667, A 0.000, B 0.000, C 0.000 }
gfCNCPoint3[17176] = {X 61.1646, Y 56.6963, Z -4.6667, A 0.000, B 0.000, C 0.000 }
gfCNCPoint3[17177] = {X 59.7147, Y 56.2224, Z -4.6667, A 0.000, B 0.000, C 0.000 }
gfCNCPoint3[17178] = {X 58.3360, Y 55.5695, Z -4.6667, A 0.000, B 0.000, C 0.000 }
gfCNCPoint3[17179] = {X 57.0507, Y 54.7481, Z -4.6667, A 0.000, B 0.000, C 0.000 }
gfCNCPoint3[17180] = {X 55.8790, Y 53.7713, Z -4.6667, A 0.000, B 0.000, C 0.000 }
gfCNCPoint3[17181] = {X 54.7074, Y 54.7481, Z -4.6667, A 0.000, B 0.000, C 0.000 }
gfCNCPoint3[17182] = {X 53.4220, Y 55.5695, Z -4.6667, A 0.000, B 0.000, C 0.000 }
gfCNCPoint3[17183] = {X 52.0434, Y 56.2224, Z -4.6667, A 0.000, B 0.000, C 0.000 }
gfCNCPoint3[17184] = {X 50.5934, Y 56.6963, Z -4.6667, A 0.000, B 0.000, C 0.000 }
gfCNCPoint3[17185] = {X 49.0953, Y 56.9837, Z -4.6667, A 0.000, B 0.000, C 0.000 }
gfCNCPoint3[17186] = {X 47.5729, Y 57.0800, Z -4.6667, A 0.000, B 0.000, C 0.000 }
gfCNCPoint3[17187] = {X 40.6393, Y 57.0800, Z -4.6667, A 0.000, B 0.000, C 0.000 }
gfCNCPoint3[17188] = {X 39.3238, Y 57.0082, Z -4.6667, A 0.000, B 0.000, C 0.000 }
gfCNCPoint3[17189] = {X 38.0239, Y 56.7935, Z -4.6667, A 0.000, B 0.000, C 0.000 }
gfCNCPoint3[17190] = {X 36.7551, Y 56.4385, Z -4.6667, A 0.000, B 0.000, C 0.000 }
gfCNCPoint3[17191] = {X 35.5326, Y 55.9475, Z -4.6667, A 0.000, B 0.000, C 0.000 }
gfCNCPoint3[17192] = {X 34.1215, Y 56.7825, Z -4.6667, A 0.000, B 0.000, C 0.000 }
gfCNCPoint3[17193] = {X 32.6341, Y 57.4725, Z -4.6667, A 0.000, B 0.000, C 0.000 }
gfCNCPoint3[17194] = {X 31.0853, Y 58.0107, Z -4.6667, A 0.000, B 0.000, C 0.000 }
gfCNCPoint3[17195] = {X 29.4906, Y 58.3917, Z -4.6667, A 0.000, B 0.000, C 0.000 }
gfCNCPoint3[17196] = {X 27.8658, Y 58.6116, Z -4.6667, A 0.000, B 0.000, C 0.000 }
gfCNCPoint3[17197] = {X 25.6557, Y 59.5459, Z -4.6667, A 0.000, B 0.000, C 0.000 }
gfCNCPoint3[17198] = {X 23.3950, Y 60.3501, Z -4.6667, A 0.000, B 0.000, C 0.000 }
gfCNCPoint3[17199] = {X 21.1538, Y 61.0054, Z -4.6667, A 0.000, B 0.000, C 0.000 }
gfCNCPoint3[17200] = {X 18.8737, Y 61.5092, Z -4.6667, A 0.000, B 0.000, C 0.000 }
gfCNCPoint3[17201] = {X 16.5651, Y 61.8592, Z -4.6667, A 0.000, B 0.000, C 0.000 }
gfCNCPoint3[17202] = {X 14.2382, Y 62.0539, Z -4.6667, A 0.000, B 0.000, C 0.000 }
gfCNCPoint3[17203] = {X 11.9034, Y 62.0923, Z -4.6667, A 0.000, B 0.000, C 0.000 }
gfCNCPoint3[17204] = {X 11.9034, Y 88.0950, Z -4.6667, A 0.000, B 0.000, C 0.000 }
gfCNCPoint3[17205] = {X 113.6337, Y 88.0950, Z -4.6667, A 0.000, B 0.000, C 0.000 }
gfCNCPoint3[17206] = {X 114.7668, Y 86.8213, Z -4.6667, A 0.000, B 0.000, C 0.000 }
gfCNCPoint3[17207] = {X 116.0418, Y 85.6896, Z -4.6667, A 0.000, B 0.000, C 0.000 }
gfCNCPoint3[17208] = {X 117.4410, Y 84.7156, Z -4.6667, A 0.000, B 0.000, C 0.000 }
gfCNCPoint3[17209] = {X 118.9449, Y 83.9127, Z -4.6667, A 0.000, B 0.000, C 0.000 }
gfCNCPoint3[17210] = {X 120.5328, Y 83.2922, Z -4.6667, A 0.000, B 0.000, C 0.000 }
gfCNCPoint3[17211] = {X 122.1826, Y 82.8627, Z -4.6667, A 0.000, B 0.000, C 0.000 }
gfCNCPoint3[17212] = {X 144.8180, Y 58.0058, Z -4.6667, A 0.000, B 0.000, C 0.000 }
gfCNCPoint3[17213] = {X 144.9144, Y 56.3317, Z -4.6667, A 0.000, B 0.000, C 0.000 }
gfCNCPoint3[17214] = {X 145.2037, Y 54.6800, Z -4.6667, A 0.000, B 0.000, C 0.000 }
gfCNCPoint3[17215] = {X 143.0396, Y 54.6800, Z -4.6667, A 0.000, B 0.000, C 0.000 }
gfCNCPoint3[17216] = {X 142.7949, Y 54.6769, Z -4.6667, A 0.000, B 0.000, C 0.000 }
gfCNCPoint3[17217] = {X 142.5504, Y 54.6676, Z -4.6667, A 0.000, B 0.000, C 0.000 }
gfCNCPoint3[17218] = {X 141.0974, Y 54.4832, Z -4.6667, A 0.000, B 0.000, C 0.000 }
gfCNCPoint3[17219] = {X 139.6889, Y 54.0816, Z -4.6667, A 0.000, B 0.000, C 0.000 }
gfCNCPoint3[17220] = {X 138.3570, Y 53.4721, Z -4.6667, A 0.000, B 0.000, C 0.000 }
gfCNCPoint3[17221] = {X 137.1324, Y 52.6686, Z -4.6667, A 0.000, B 0.000, C 0.000 }
gfCNCPoint3[17222] = {X 136.0430, Y 51.6896, Z -4.6667, A 0.000, B 0.000, C 0.000 }
gfCNCPoint3[17223] = {X 135.1138, Y 50.5574, Z -4.6667, A 0.000, B 0.000, C 0.000 }
gfCNCPoint3[17224] = {X 134.3661, Y 49.2980, Z -4.6667, A 0.000, B 0.000, C 0.000 }
gfCNCPoint3[17225] = {X 133.8169, Y 47.9401, Z -4.6667, A 0.000, B 0.000, C 0.000 }
gfCNCPoint3[17226] = {X 133.4789, Y 46.5150, Z -4.6667, A 0.000, B 0.000, C 0.000 }
gfCNCPoint3[17227] = {X 133.3598, Y 45.0552, Z -4.6667, A 0.000, B 0.000, C 0.000 }
gfCNCPoint3[17228] = {X 133.3601, Y 44.1104, Z -4.6667, A 0.000, B 0.000, C 0.000 }
gfCNCPoint3[17229] = {X 133.4665, Y 42.7742, Z -4.6667, A 0.000, B 0.000, C 0.000 }
gfCNCPoint3[17230] = {X 133.7565, Y 41.4655, Z -4.6667, A 0.000, B 0.000, C 0.000 }
gfCNCPoint3[17231] = {X 136.0581, Y 42.1457, Z -4.6667, A 0.000, B 0.000, C 0.000 }
gfCNCPoint3[17232] = {X 136.3664, Y 41.2990, Z -4.6667, A 0.000, B 0.000, C 0.000 }
gfCNCPoint3[17233] = {X 136.7770, Y 40.4969, Z -4.6667, A 0.000, B 0.000, C 0.000 }
gfCNCPoint3[17234] = {X 137.2836, Y 39.7516, Z -4.6667, A 0.000, B 0.000, C 0.000 }
gfCNCPoint3[17235] = {X 137.2836, Y 23.8768, Z -4.6667, A 0.000, B 0.000, C 0.000 }
gfCNCPoint3[17236] = {X 136.4352, Y 24.2641, Z -4.6667, A 0.000, B 0.000, C 0.000 }
gfCNCPoint3[17237] = {X 135.5443, Y 24.5398, Z -4.6667, A 0.000, B 0.000, C 0.000 }
gfCNCPoint3[17238] = {X 134.6254, Y 24.6993, Z -4.6667, A 0.000, B 0.000, C 0.000 }
gfCNCPoint3[17239] = {X 134.2595, Y 24.7296, Z -4.6667, A 0.000, B 0.000, C 0.000 }
gfCNCPoint3[17240] = {X 133.8926, Y 24.7414, Z -4.6667, A 0.000, B 0.000, C 0.000 }
gfCNCPoint3[17241] = {X 133.2006, Y 24.7415, Z -4.6667, A 0.000, B 0.000, C 0.000 }
gfCNCPoint3[17242] = {X 131.9931, Y 24.6407, Z -4.6667, A 0.000, B 0.000, C 0.000 }
gfCNCPoint3[17243] = {X 130.8190, Y 24.3410, Z -4.6667, A 0.000, B 0.000, C 0.000 }
gfCNCPoint3[17244] = {X 129.7109, Y 23.8506, Z -4.6667, A 0.000, B 0.000, C 0.000 }
gfCNCPoint3[17245] = {X 128.6995, Y 23.1833, Z -4.6667, A 0.000, B 0.000, C 0.000 }
gfCNCPoint3[17246] = {X 127.8128, Y 22.3574, Z -4.6667, A 0.000, B 0.000, C 0.000 }
gfCNCPoint3[17247] = {X 127.0754, Y 21.3959, Z -4.6667, A 0.000, B 0.000, C 0.000 }
gfCNCPoint3[17248] = {X 126.5076, Y 20.3254, Z -4.6667, A 0.000, B 0.000, C 0.000 }
gfCNCPoint3[17249] = {X 126.1253, Y 19.1756, Z -4.6667, A 0.000, B 0.000, C 0.000 }
gfCNCPoint3[17250] = {X 125.9390, Y 17.9783, Z -4.6667, A 0.000, B 0.000, C 0.000 }
gfCNCPoint3[17251] = {X 125.9252, Y 17.7201, Z -4.6667, A 0.000, B 0.000, C 0.000 }
gfCNCPoint3[17252] = {X 125.9206, Y 17.4615, Z -4.6667, A 0.000, B 0.000, C 0.000 }
gfCNCPoint3[17253] = {X 125.9206, Y 10.4835, Z -4.6667, A 0.000, B 0.000, C 0.000 }
gfCNCPoint3[17254] = {X 125.9372, Y 9.9931, Z -4.6667, A 0.000, B 0.000, C 0.000 }
gfCNCPoint3[17255] = {X 125.9867, Y 9.5050, Z -4.6667, A 0.000, B 0.000, C 0.000 }
gfCNCPoint3[17256] = {X 121.8686, Y 9.5050, Z -4.6667, A 0.000, B 0.000, C 0.000 }
gfCNCPoint3[17257] = {X 122.3090, Y 10.3410, Z -4.6667, A 0.000, B 0.000, C 0.000 }
gfCNCPoint3[17258] = {X 122.5801, Y 11.2463, Z -4.6667, A 0.000, B 0.000, C 0.000 }
gfCNCPoint3[17259] = {X 122.6716, Y 12.1868, Z -4.6667, A 0.000, B 0.000, C 0.000 }
gfCNCPoint3[17260] = {X 122.6714, Y 13.0237, Z -4.6667, A 0.000, B 0.000, C 0.000 }
gfCNCPoint3[17261] = {X 122.5640, Y 13.9968, Z -4.6667, A 0.000, B 0.000, C 0.000 }
gfCNCPoint3[17262] = {X 122.2647, Y 14.9289, Z -4.6667, A 0.000, B 0.000, C 0.000 }
gfCNCPoint3[17263] = {X 121.7853, Y 15.7825, Z -4.6667, A 0.000, B 0.000, C 0.000 }
gfCNCPoint3[17264] = {X 121.1451, Y 16.5232, Z -4.6667, A 0.000, B 0.000, C 0.000 }
gfCNCPoint3[17265] = {X 121.1441, Y 40.6626, Z -4.6667, A 0.000, B 0.000, C 0.000 }
gfCNCPoint3[17266] = {X 121.7854, Y 41.4046, Z -4.6667, A 0.000, B 0.000, C 0.000 }
gfCNCPoint3[17267] = {X 122.2655, Y 42.2599, Z -4.6667, A 0.000, B 0.000, C 0.000 }
gfCNCPoint3[17268] = {X 122.5649, Y 43.1938, Z -4.6667, A 0.000, B 0.000, C 0.000 }
gfCNCPoint3[17269] = {X 122.6714, Y 44.1688, Z -4.6667, A 0.000, B 0.000, C 0.000 }
gfCNCPoint3[17270] = {X 122.6716, Y 45.0000, Z -4.6667, A 0.000, B 0.000, C 0.000 }
gfCNCPoint3[17271] = {X 122.5778, Y 45.9520, Z -4.6667, A 0.000, B 0.000, C 0.000 }
gfCNCPoint3[17272] = {X 122.3001, Y 46.8675, Z -4.6667, A 0.000, B 0.000, C 0.000 }
gfCNCPoint3[17273] = {X 121.8491, Y 47.7112, Z -4.6667, A 0.000, B 0.000, C 0.000 }
gfCNCPoint3[17274] = {X 121.2423, Y 48.4507, Z -4.6667, A 0.000, B 0.000, C 0.000 }
gfCNCPoint3[17275] = {X 120.5028, Y 49.0576, Z -4.6667, A 0.000, B 0.000, C 0.000 }
gfCNCPoint3[17276] = {X 119.6591, Y 49.5085, Z -4.6667, A 0.000, B 0.000, C 0.000 }
gfCNCPoint3[17277] = {X 118.7436, Y 49.7862, Z -4.6667, A 0.000, B 0.000, C 0.000 }
gfCNCPoint3[17278] = {X 117.7916, Y 49.8800, Z -4.6667, A 0.000, B 0.000, C 0.000 }
gfCNCPoint3[17279] = {X 111.9185, Y 49.8800, Z -4.6667, A 0.000, B 0.000, C 0.000 }
gfCNCPoint3[17280] = {X 111.0234, Y 49.7972, Z -4.6667, A 0.000, B 0.000, C 0.000 }
gfCNCPoint3[17281] = {X 110.1587, Y 49.5517, Z -4.6667, A 0.000, B 0.000, C 0.000 }
gfCNCPoint3[17282] = {X 109.3537, Y 49.1517, Z -4.6667, A 0.000, B 0.000, C 0.000 }
gfCNCPoint3[17283] = {X 108.6357, Y 48.6108, Z -4.6667, A 0.000, B 0.000, C 0.000 }
gfCNCPoint3[17284] = {X 108.0714, Y 48.0024, Z -4.6667, A 0.000, B 0.000, C 0.000 }
gfCNCPoint3[17285] = {X 107.6183, Y 47.3071, Z -4.6667, A 0.000, B 0.000, C 0.000 }
gfCNCPoint3[17286] = {X 107.2895, Y 46.5451, Z -4.6667, A 0.000, B 0.000, C 0.000 }
gfCNCPoint3[17287] = {X 107.0947, Y 45.7384, Z -4.6667, A 0.000, B 0.000, C 0.000 }
gfCNCPoint3[17288] = {X 106.6287, Y 46.8769, Z -4.6667, A 0.000, B 0.000, C 0.000 }
gfCNCPoint3[17289] = {X 106.1131, Y 47.8110, Z -4.6667, A 0.000, B 0.000, C 0.000 }
gfCNCPoint3[17290] = {X 105.4068, Y 48.6108, Z -4.6667, A 0.000, B 0.000, C 0.000 }
gfCNCPoint3[17291] = {X 104.8391, Y 49.0550, Z -4.6667, A 0.000, B 0.000, C 0.000 }
gfCNCPoint3[17292] = {X 104.2121, Y 49.4107, Z -4.6667, A 0.000, B 0.000, C 0.000 }
gfCNCPoint3[17293] = {X 103.3106, Y 49.7335, Z -4.6667, A 0.000, B 0.000, C 0.000 }
gfCNCPoint3[17294] = {X 102.3635, Y 49.8741, Z -4.6667, A 0.000, B 0.000, C 0.000 }
gfCNCPoint3[17295] = {X 101.4071, Y 49.8271, Z -4.6667, A 0.000, B 0.000, C 0.000 }
gfCNCPoint3[17296] = {X 100.4784, Y 49.5941, Z -4.6667, A 0.000, B 0.000, C 0.000 }
gfCNCPoint3[17297] = {X 99.6130, Y 49.1844, Z -4.6667, A 0.000, B 0.000, C 0.000 }
gfCNCPoint3[17298] = {X 98.8443, Y 48.6135, Z -4.6667, A 0.000, B 0.000, C 0.000 }
gfCNCPoint3[17299] = {X 98.1362, Y 47.8127, Z -4.6667, A 0.000, B 0.000, C 0.000 }
gfCNCPoint3[17300] = {X 97.6194, Y 46.8769, Z -4.6667, A 0.000, B 0.000, C 0.000 }
gfCNCPoint3[17301] = {X 97.1600, Y 45.7536, Z -4.6667, A 0.000, B 0.000, C 0.000 }
gfCNCPoint3[17302] = {X 96.9635, Y 46.5570, Z -4.6667, A 0.000, B 0.000, C 0.000 }
gfCNCPoint3[17303] = {X 96.6342, Y 47.3156, Z -4.6667, A 0.000, B 0.000, C 0.000 }
gfCNCPoint3[17304] = {X 96.1814, Y 48.0078, Z -4.6667, A 0.000, B 0.000, C 0.000 }
gfCNCPoint3[17305] = {X 95.6183, Y 48.6135, Z -4.6667, A 0.000, B 0.000, C 0.000 }
gfCNCPoint3[17306] = {X 94.9007, Y 49.1533, Z -4.6667, A 0.000, B 0.000, C 0.000 }
gfCNCPoint3[17307] = {X 94.0964, Y 49.5524, Z -4.6667, A 0.000, B 0.000, C 0.000 }
gfCNCPoint3[17308] = {X 93.2326, Y 49.7974, Z -4.6667, A 0.000, B 0.000, C 0.000 }
gfCNCPoint3[17309] = {X 92.3385, Y 49.8800, Z -4.6667, A 0.000, B 0.000, C 0.000 }
gfCNCPoint3[17310] = {X 85.8951, Y 49.8800, Z -4.6667, A 0.000, B 0.000, C 0.000 }
gfCNCPoint3[17311] = {X 85.0841, Y 49.8121, Z -4.6667, A 0.000, B 0.000, C 0.000 }
gfCNCPoint3[17312] = {X 84.2956, Y 49.6104, Z -4.6667, A 0.000, B 0.000, C 0.000 }
gfCNCPoint3[17313] = {X 83.5517, Y 49.2805, Z -4.6667, A 0.000, B 0.000, C 0.000 }
gfCNCPoint3[17314] = {X 82.8729, Y 48.8316, Z -4.6667, A 0.000, B 0.000, C 0.000 }
gfCNCPoint3[17315] = {X 82.2391, Y 48.2324, Z -4.6667, A 0.000, B 0.000, C 0.000 }
gfCNCPoint3[17316] = {X 81.7221, Y 47.5300, Z -4.6667, A 0.000, B 0.000, C 0.000 }
gfCNCPoint3[17317] = {X 81.3384, Y 46.7467, Z -4.6667, A 0.000, B 0.000, C 0.000 }
gfCNCPoint3[17318] = {X 81.1002, Y 45.9077, Z -4.6667, A 0.000, B 0.000, C 0.000 }
gfCNCPoint3[17319] = {X 81.0152, Y 45.0397, Z -4.6667, A 0.000, B 0.000, C 0.000 }
gfCNCPoint3[17320] = {X 81.0151, Y 44.2038, Z -4.6667, A 0.000, B 0.000, C 0.000 }
gfCNCPoint3[17321] = {X 81.1199, Y 43.2201, Z -4.6667, A 0.000, B 0.000, C 0.000 }
gfCNCPoint3[17322] = {X 81.4186, Y 42.2770, Z -4.6667, A 0.000, B 0.000, C 0.000 }
gfCNCPoint3[17323] = {X 81.8994, Y 41.4123, Z -4.6667, A 0.000, B 0.000, C 0.000 }
gfCNCPoint3[17324] = {X 82.5428, Y 40.6609, Z -4.6667, A 0.000, B 0.000, C 0.000 }
gfCNCPoint3[17325] = {X 82.5425, Y 16.5241, Z -4.6667, A 0.000, B 0.000, C 0.000 }
gfCNCPoint3[17326] = {X 81.9014, Y 15.7825, Z -4.6667, A 0.000, B 0.000, C 0.000 }
gfCNCPoint3[17327] = {X 81.4214, Y 14.9276, Z -4.6667, A 0.000, B 0.000, C 0.000 }
gfCNCPoint3[17328] = {X 81.1220, Y 13.9941, Z -4.6667, A 0.000, B 0.000, C 0.000 }
gfCNCPoint3[17329] = {X 81.0153, Y 13.0196, Z -4.6667, A 0.000, B 0.000, C 0.000 }
gfCNCPoint3[17330] = {X 81.0151, Y 12.1868, Z -4.6667, A 0.000, B 0.000, C 0.000 }
gfCNCPoint3[17331] = {X 81.0160, Y 12.0923, Z -4.6667, A 0.000, B 0.000, C 0.000 }
gfCNCPoint3[17332] = {X 81.0187, Y 11.9979, Z -4.6667, A 0.000, B 0.000, C 0.000 }
gfCNCPoint3[17333] = {X 81.1324, Y 11.1230, Z -4.6667, A 0.000, B 0.000, C 0.000 }
gfCNCPoint3[17334] = {X 81.4018, Y 10.2829, Z -4.6667, A 0.000, B 0.000, C 0.000 }
gfCNCPoint3[17335] = {X 81.8181, Y 9.5050, Z -4.6667, A 0.000, B 0.000, C 0.000 }
gfCNCPoint3[17336] = {X 82.2191, Y 9.7688, Z -4.6667, A 0.000, B 0.000, C 0.000 }
gfCNCPoint3[17337] = {X 82.7659, Y 9.0936, Z -4.6667, A 0.000, B 0.000, C 0.000 }
gfCNCPoint3[17338] = {X 83.4348, Y 8.5390, Z -4.6667, A 0.000, B 0.000, C 0.000 }
gfCNCPoint3[17339] = {X 84.1995, Y 8.1266, Z -4.6667, A 0.000, B 0.000, C 0.000 }
gfCNCPoint3[17340] = {X 85.0305, Y 7.8726, Z -4.6667, A 0.000, B 0.000, C 0.000 }
gfCNCPoint3[17341] = {X 85.8951, Y 7.7868, Z -4.6667, A 0.000, B 0.000, C 0.000 }
gfCNCPoint3[17342] = {X 94.0497, Y 7.7868, Z -4.6667, A 0.000, B 0.000, C 0.000 }
gfCNCPoint3[17343] = {X 95.0288, Y 7.8971, Z -4.6667, A 0.000, B 0.000, C 0.000 }
gfCNCPoint3[17344] = {X 95.9588, Y 8.2226, Z -4.6667, A 0.000, B 0.000, C 0.000 }
gfCNCPoint3[17345] = {X 96.7930, Y 8.7468, Z -4.6667, A 0.000, B 0.000, C 0.000 }
gfCNCPoint3[17346] = {X 97.4897, Y 9.4435, Z -4.6667, A 0.000, B 0.000, C 0.000 }
gfCNCPoint3[17347] = {X 98.0139, Y 10.2777, Z -4.6667, A 0.000, B 0.000, C 0.000 }
gfCNCPoint3[17348] = {X 98.3394, Y 11.2077, Z -4.6667, A 0.000, B 0.000, C 0.000 }
gfCNCPoint3[17349] = {X 98.4497, Y 12.1868, Z -4.6667, A 0.000, B 0.000, C 0.000 }
gfCNCPoint3[17350] = {X 98.4494, Y 13.0233, Z -4.6667, A 0.000, B 0.000, C 0.000 }
gfCNCPoint3[17351] = {X 98.3724, Y 13.7991, Z -4.6667, A 0.000, B 0.000, C 0.000 }
gfCNCPoint3[17352] = {X 98.1596, Y 14.5492, Z -4.6667, A 0.000, B 0.000, C 0.000 }
gfCNCPoint3[17353] = {X 97.8178, Y 15.2499, Z -4.6667, A 0.000, B 0.000, C 0.000 }
gfCNCPoint3[17354] = {X 98.3679, Y 16.6194, Z -4.6667, A 0.000, B 0.000, C 0.000 }
gfCNCPoint3[17355] = {X 101.8765, Y 25.3167, Z -4.6667, A 0.000, B 0.000, C 0.000 }
gfCNCPoint3[17356] = {X 105.9240, Y 15.2228, Z -4.6667, A 0.000, B 0.000, C 0.000 }
gfCNCPoint3[17357] = {X 105.5856, Y 14.5154, Z -4.6667, A 0.000, B 0.000, C 0.000 }
gfCNCPoint3[17358] = {X 105.3782, Y 13.7591, Z -4.6667, A 0.000, B 0.000, C 0.000 }
gfCNCPoint3[17359] = {X 105.3083, Y 12.9779, Z -4.6667, A 0.000, B 0.000, C 0.000 }
gfCNCPoint3[17360] = {X 105.3083, Y 12.1868, Z -4.6667, A 0.000, B 0.000, C 0.000 }
gfCNCPoint3[17361] = {X 105.4186, Y 11.2077, Z -4.6667, A 0.000, B 0.000, C 0.000 }
gfCNCPoint3[17362] = {X 105.7440, Y 10.2777, Z -4.6667, A 0.000, B 0.000, C 0.000 }
gfCNCPoint3[17363] = {X 106.2682, Y 9.4435, Z -4.6667, A 0.000, B 0.000, C 0.000 }
gfCNCPoint3[17364] = {X 106.9649, Y 8.7468, Z -4.6667, A 0.000, B 0.000, C 0.000 }
gfCNCPoint3[17365] = {X 107.7992, Y 8.2226, Z -4.6667, A 0.000, B 0.000, C 0.000 }
gfCNCPoint3[17366] = {X 108.7292, Y 7.8971, Z -4.6667, A 0.000, B 0.000, C 0.000 }
gfCNCPoint3[17367] = {X 109.7083, Y 7.7868, Z -4.6667, A 0.000, B 0.000, C 0.000 }
gfCNCPoint3[17368] = {X 117.7916, Y 7.7868, Z -4.6667, A 0.000, B 0.000, C 0.000 }
gfCNCPoint3[17369] = {X 118.7707, Y 7.8971, Z -4.6667, A 0.000, B 0.000, C 0.000 }
gfCNCPoint3[17370] = {X 119.7007, Y 8.2226, Z -4.6667, A 0.000, B 0.000, C 0.000 }
gfCNCPoint3[17371] = {X 120.5349, Y 8.7468, Z -4.6667, A 0.000, B 0.000, C 0.000 }
gfCNCPoint3[17372] = {X 121.2316, Y 9.4435, Z -4.6667, A 0.000, B 0.000, C 0.000 }
gfCNCPoint3[17373] = {X 121.7558, Y 10.2777, Z -4.6667, A 0.000, B 0.000, C 0.000 }
gfCNCPoint3[17374] = {X 122.0813, Y 11.2077, Z -4.6667, A 0.000, B 0.000, C 0.000 }
gfCNCPoint3[17375] = {X 122.1916, Y 12.1868, Z -4.6667, A 0.000, B 0.000, C 0.000 }
gfCNCPoint3[17376] = {X 122.1913, Y 13.0233, Z -4.6667, A 0.000, B 0.000, C 0.000 }
gfCNCPoint3[17377] = {X 122.0831, Y 13.9490, Z -4.6667, A 0.000, B 0.000, C 0.000 }
gfCNCPoint3[17378] = {X 121.7823, Y 14.8311, Z -4.6667, A 0.000, B 0.000, C 0.000 }
gfCNCPoint3[17379] = {X 121.3025, Y 15.6301, Z -4.6667, A 0.000, B 0.000, C 0.000 }
gfCNCPoint3[17380] = {X 120.6651, Y 16.3101, Z -4.6667, A 0.000, B 0.000, C 0.000 }
gfCNCPoint3[17381] = {X 120.6641, Y 40.8763, Z -4.6667, A 0.000, B 0.000, C 0.000 }
gfCNCPoint3[17382] = {X 120.6784, Y 40.8882, Z -4.6667, A 0.000, B 0.000, C 0.000 }
gfCNCPoint3[17383] = {X 121.3172, Y 41.5763, Z -4.6667, A 0.000, B 0.000, C 0.000 }
gfCNCPoint3[17384] = {X 121.7955, Y 42.3843, Z -4.6667, A 0.000, B 0.000, C 0.000 }
gfCNCPoint3[17385] = {X 122.0914, Y 43.2753, Z -4.6667, A 0.000, B 0.000, C 0.000 }
gfCNCPoint3[17386] = {X 122.1916, Y 44.2089, Z -4.6667, A 0.000, B 0.000, C 0.000 }
gfCNCPoint3[17387] = {X 122.1916, Y 45.0000, Z -4.6667, A 0.000, B 0.000, C 0.000 }
gfCNCPoint3[17388] = {X 122.0813, Y 45.9791, Z -4.6667, A 0.000, B 0.000, C 0.000 }
gfCNCPoint3[17389] = {X 121.7558, Y 46.9091, Z -4.6667, A 0.000, B 0.000, C 0.000 }
gfCNCPoint3[17390] = {X 121.2316, Y 47.7434, Z -4.6667, A 0.000, B 0.000, C 0.000 }
gfCNCPoint3[17391] = {X 120.5349, Y 48.4401, Z -4.6667, A 0.000, B 0.000, C 0.000 }
gfCNCPoint3[17392] = {X 119.7007, Y 48.9643, Z -4.6667, A 0.000, B 0.000, C 0.000 }
gfCNCPoint3[17393] = {X 118.7707, Y 49.2897, Z -4.6667, A 0.000, B 0.000, C 0.000 }
gfCNCPoint3[17394] = {X 117.7916, Y 49.4000, Z -4.6667, A 0.000, B 0.000, C 0.000 }
gfCNCPoint3[17395] = {X 111.9185, Y 49.4000, Z -4.6667, A 0.000, B 0.000, C 0.000 }
gfCNCPoint3[17396] = {X 110.9394, Y 49.2897, Z -4.6667, A 0.000, B 0.000, C 0.000 }
gfCNCPoint3[17397] = {X 110.0094, Y 48.9643, Z -4.6667, A 0.000, B 0.000, C 0.000 }
gfCNCPoint3[17398] = {X 109.1751, Y 48.4400, Z -4.6667, A 0.000, B 0.000, C 0.000 }
gfCNCPoint3[17399] = {X 108.4784, Y 47.7433, Z -4.6667, A 0.000, B 0.000, C 0.000 }
gfCNCPoint3[17400] = {X 107.9542, Y 46.9091, Z -4.6667, A 0.000, B 0.000, C 0.000 }
gfCNCPoint3[17401] = {X 107.6288, Y 45.9791, Z -4.6667, A 0.000, B 0.000, C 0.000 }
gfCNCPoint3[17402] = {X 107.5185, Y 45.0000, Z -4.6667, A 0.000, B 0.000, C 0.000 }
gfCNCPoint3[17403] = {X 107.5185, Y 44.1775, Z -4.6667, A 0.000, B 0.000, C 0.000 }
gfCNCPoint3[17404] = {X 107.5547, Y 43.6256, Z -4.6667, A 0.000, B 0.000, C 0.000 }
gfCNCPoint3[17405] = {X 107.6626, Y 43.0832, Z -4.6667, A 0.000, B 0.000, C 0.000 }
gfCNCPoint3[17406] = {X 106.1856, Y 46.6923, Z -4.6667, A 0.000, B 0.000, C 0.000 }
gfCNCPoint3[17407] = {X 105.8087, Y 47.4049, Z -4.6667, A 0.000, B 0.000, C 0.000 }
gfCNCPoint3[17408] = {X 105.3081, Y 48.0367, Z -4.6667, A 0.000, B 0.000, C 0.000 }
gfCNCPoint3[17409] = {X 104.7006, Y 48.5667, Z -4.6667, A 0.000, B 0.000, C 0.000 }
gfCNCPoint3[17410] = {X 104.0067, Y 48.9769, Z -4.6667, A 0.000, B 0.000, C 0.000 }
gfCNCPoint3[17411] = {X 103.0414, Y 49.3033, Z -4.6667, A 0.000, B 0.000, C 0.000 }
gfCNCPoint3[17412] = {X 102.0269, Y 49.3989, Z -4.6667, A 0.000, B 0.000, C 0.000 }
gfCNCPoint3[17413] = {X 101.0176, Y 49.2586, Z -4.6667, A 0.000, B 0.000, C 0.000 }
gfCNCPoint3[17414] = {X 100.0676, Y 48.8899, Z -4.6667, A 0.000, B 0.000, C 0.000 }
gfCNCPoint3[17415] = {X 99.2280, Y 48.3125, Z -4.6667, A 0.000, B 0.000, C 0.000 }
gfCNCPoint3[17416] = {X 98.5436, Y 47.5575, Z -4.6667, A 0.000, B 0.000, C 0.000 }
gfCNCPoint3[17417] = {X 98.0514, Y 46.6653, Z -4.6667, A 0.000, B 0.000, C 0.000 }
gfCNCPoint3[17418] = {X 96.5874, Y 43.0848, Z -4.6667, A 0.000, B 0.000, C 0.000 }
gfCNCPoint3[17419] = {X 96.6986, Y 43.6421, Z -4.6667, A 0.000, B 0.000, C 0.000 }
gfCNCPoint3[17420] = {X 96.7385, Y 44.2089, Z -4.6667, A 0.000, B 0.000, C 0.000 }
gfCNCPoint3[17421] = {X 96.7383, Y 45.0423, Z -4.6667, A 0.000, B 0.000, C 0.000 }
gfCNCPoint3[17422] = {X 96.6200, Y 46.0144, Z -4.6667, A 0.000, B 0.000, C 0.000 }
gfCNCPoint3[17423] = {X 96.2896, Y 46.9363, Z -4.6667, A 0.000, B 0.000, C 0.000 }
gfCNCPoint3[17424] = {X 95.7635, Y 47.7622, Z -4.6667, A 0.000, B 0.000, C 0.000 }
gfCNCPoint3[17425] = {X 95.0677, Y 48.4513, Z -4.6667, A 0.000, B 0.000, C 0.000 }
gfCNCPoint3[17426] = {X 94.2367, Y 48.9695, Z -4.6667, A 0.000, B 0.000, C 0.000 }
gfCNCPoint3[17427] = {X 93.3117, Y 49.2910, Z -4.6667, A 0.000, B 0.000, C 0.000 }
gfCNCPoint3[17428] = {X 92.3385, Y 49.4000, Z -4.6667, A 0.000, B 0.000, C 0.000 }
gfCNCPoint3[17429] = {X 85.8951, Y 49.4000, Z -4.6667, A 0.000, B 0.000, C 0.000 }
gfCNCPoint3[17430] = {X 84.9160, Y 49.2897, Z -4.6667, A 0.000, B 0.000, C 0.000 }
gfCNCPoint3[17431] = {X 83.9860, Y 48.9643, Z -4.6667, A 0.000, B 0.000, C 0.000 }
gfCNCPoint3[17432] = {X 83.1517, Y 48.4400, Z -4.6667, A 0.000, B 0.000, C 0.000 }
gfCNCPoint3[17433] = {X 82.4550, Y 47.7433, Z -4.6667, A 0.000, B 0.000, C 0.000 }
gfCNCPoint3[17434] = {X 81.9308, Y 46.9091, Z -4.6667, A 0.000, B 0.000, C 0.000 }
gfCNCPoint3[17435] = {X 81.6054, Y 45.9791, Z -4.6667, A 0.000, B 0.000, C 0.000 }
gfCNCPoint3[17436] = {X 81.4951, Y 45.0000, Z -4.6667, A 0.000, B 0.000, C 0.000 }
gfCNCPoint3[17437] = {X 81.4951, Y 44.2066, Z -4.6667, A 0.000, B 0.000, C 0.000 }
gfCNCPoint3[17438] = {X 81.6003, Y 43.2693, Z -4.6667, A 0.000, B 0.000, C 0.000 }
gfCNCPoint3[17439] = {X 81.9002, Y 42.3752, Z -4.6667, A 0.000, B 0.000, C 0.000 }
gfCNCPoint3[17440] = {X 82.3816, Y 41.5641, Z -4.6667, A 0.000, B 0.000, C 0.000 }
gfCNCPoint3[17441] = {X 83.0228, Y 40.8725, Z -4.6667, A 0.000, B 0.000, C 0.000 }
gfCNCPoint3[17442] = {X 83.0225, Y 16.3109, Z -4.6667, A 0.000, B 0.000, C 0.000 }
gfCNCPoint3[17443] = {X 82.3779, Y 15.6218, Z -4.6667, A 0.000, B 0.000, C 0.000 }
gfCNCPoint3[17444] = {X 81.8951, Y 14.8111, Z -4.6667, A 0.000, B 0.000, C 0.000 }
gfCNCPoint3[17445] = {X 81.5962, Y 13.9161, Z -4.6667, A 0.000, B 0.000, C 0.000 }
gfCNCPoint3[17446] = {X 81.4951, Y 12.9779, Z -4.6667, A 0.000, B 0.000, C 0.000 }
gfCNCPoint3[17447] = {X 81.4951, Y 12.1868, Z -4.6667, A 0.000, B 0.000, C 0.000 }
gfCNCPoint3[17448] = {X 81.5776, Y 11.3388, Z -4.6667, A 0.000, B 0.000, C 0.000 }
gfCNCPoint3[17449] = {X 81.8220, Y 10.5226, Z -4.6667, A 0.000, B 0.000, C 0.000 }
gfCNCPoint3[17450] = {X 82.2191, Y 9.7688, Z -4.6667, A 0.000, B 0.000, C 0.000 }
gfCNCPoint3[17451] = {X 81.8181, Y 9.5050, Z -4.6667, A 0.000, B 0.000, C 0.000 }
gfCNCPoint3[17452] = {X 68.9232, Y 9.5050, Z -4.6667, A 0.000, B 0.000, C 0.000 }
gfCNCPoint3[17453] = {X 69.1905, Y 10.7208, Z -4.6667, A 0.000, B 0.000, C 0.000 }
gfCNCPoint3[17454] = {X 69.2995, Y 11.9610, Z -4.6667, A 0.000, B 0.000, C 0.000 }
gfCNCPoint3[17455] = {X 69.3015, Y 12.0739, Z -4.6667, A 0.000, B 0.000, C 0.000 }
gfCNCPoint3[17456] = {X 69.3021, Y 12.1868, Z -4.6667, A 0.000, B 0.000, C 0.000 }
gfCNCPoint3[17457] = {X 69.3017, Y 13.0686, Z -4.6667, A 0.000, B 0.000, C 0.000 }
gfCNCPoint3[17458] = {X 69.2127, Y 14.2906, Z -4.6667, A 0.000, B 0.000, C 0.000 }
gfCNCPoint3[17459] = {X 68.9701, Y 15.4915, Z -4.6667, A 0.000, B 0.000, C 0.000 }
gfCNCPoint3[17460] = {X 73.2465, Y 26.9311, Z -4.6667, A 0.000, B 0.000, C 0.000 }
gfCNCPoint3[17461] = {X 77.7426, Y 25.2503, Z -4.6667, A 0.000, B 0.000, C 0.000 }
gfCNCPoint3[17462] = {X 77.7425, Y 18.1971, Z -4.6667, A 0.000, B 0.000, C 0.000 }
gfCNCPoint3[17463] = {X 77.0781, Y 16.9734, Z -4.6667, A 0.000, B 0.000, C 0.000 }
gfCNCPoint3[17464] = {X 76.5960, Y 15.6670, Z -4.6667, A 0.000, B 0.000, C 0.000 }
gfCNCPoint3[17465] = {X 76.3065, Y 14.3050, Z -4.6667, A 0.000, B 0.000, C 0.000 }
gfCNCPoint3[17466] = {X 74.0412, Y 14.3050, Z -4.6667, A 0.000, B 0.000, C 0.000 }
gfCNCPoint3[17467] = {X 73.9993, Y 14.7009, Z -4.6667, A 0.000, B 0.000, C 0.000 }
gfCNCPoint3[17468] = {X 73.9465, Y 15.0955, Z -4.6667, A 0.000, B 0.000, C 0.000 }
gfCNCPoint3[17469] = {X 77.7426, Y 25.2503, Z -4.6667, A 0.000, B 0.000, C 0.000 }
gfCNCPoint3[17470] = {X 75.4946, Y 26.0907, Z -4.6667, A 0.000, B 0.000, C 0.000 }
gfCNCPoint3[17471] = {X 78.9553, Y 35.3483, Z -4.6667, A 0.000, B 0.000, C 0.000 }
gfCNCPoint3[17472] = {X 79.5719, Y 35.9624, Z -4.6667, A 0.000, B 0.000, C 0.000 }
gfCNCPoint3[17473] = {X 80.1427, Y 36.6194, Z -4.6667, A 0.000, B 0.000, C 0.000 }
gfCNCPoint3[17474] = {X 80.1425, Y 17.4397, Z -4.6667, A 0.000, B 0.000, C 0.000 }
gfCNCPoint3[17475] = {X 79.4943, Y 16.4462, Z -4.6667, A 0.000, B 0.000, C 0.000 }
gfCNCPoint3[17476] = {X 79.0160, Y 15.3606, Z -4.6667, A 0.000, B 0.000, C 0.000 }
gfCNCPoint3[17477] = {X 78.7204, Y 14.2117, Z -4.6667, A 0.000, B 0.000, C 0.000 }
gfCNCPoint3[17478] = {X 78.6153, Y 13.0301, Z -4.6667, A 0.000, B 0.000, C 0.000 }
gfCNCPoint3[17479] = {X 78.6151, Y 12.1868, Z -4.6667, A 0.000, B 0.000, C 0.000 }
gfCNCPoint3[17480] = {X 78.6164, Y 12.0459, Z -4.6667, A 0.000, B 0.000, C 0.000 }
gfCNCPoint3[17481] = {X 78.6205, Y 11.9050, Z -4.6667, A 0.000, B 0.000, C 0.000 }
gfCNCPoint3[17482] = {X 71.6988, Y 11.9050, Z -4.6667, A 0.000, B 0.000, C 0.000 }
gfCNCPoint3[17483] = {X 71.7013, Y 12.0459, Z -4.6667, A 0.000, B 0.000, C 0.000 }
gfCNCPoint3[17484] = {X 71.7021, Y 12.1868, Z -4.6667, A 0.000, B 0.000, C 0.000 }
gfCNCPoint3[17485] = {X 71.7016, Y 13.0911, Z -4.6667, A 0.000, B 0.000, C 0.000 }
gfCNCPoint3[17486] = {X 71.6386, Y 14.2151, Z -4.6667, A 0.000, B 0.000, C 0.000 }
gfCNCPoint3[17487] = {X 71.4713, Y 15.3283, Z -4.6667, A 0.000, B 0.000, C 0.000 }
gfCNCPoint3[17488] = {X 75.4946, Y 26.0907, Z -4.6667, A 0.000, B 0.000, C 0.000 }
gfCNCPoint3[17489] = {X 73.2465, Y 26.9311, Z -4.6667, A 0.000, B 0.000, C 0.000 }
gfCNCPoint3[17490] = {X 76.9182, Y 36.7531, Z -4.6667, A 0.000, B 0.000, C 0.000 }
gfCNCPoint3[17491] = {X 77.6312, Y 37.4062, Z -4.6667, A 0.000, B 0.000, C 0.000 }
gfCNCPoint3[17492] = {X 78.2755, Y 38.1272, Z -4.6667, A 0.000, B 0.000, C 0.000 }
gfCNCPoint3[17493] = {X 79.0231, Y 39.1921, Z -4.6667, A 0.000, B 0.000, C 0.000 }
gfCNCPoint3[17494] = {X 79.6210, Y 40.3476, Z -4.6667, A 0.000, B 0.000, C 0.000 }
gfCNCPoint3[17495] = {X 80.0587, Y 41.5728, Z -4.6667, A 0.000, B 0.000, C 0.000 }
gfCNCPoint3[17496] = {X 80.3280, Y 42.8457, Z -4.6667, A 0.000, B 0.000, C 0.000 }
gfCNCPoint3[17497] = {X 80.4242, Y 44.1432, Z -4.6667, A 0.000, B 0.000, C 0.000 }
gfCNCPoint3[17498] = {X 80.4245, Y 45.0000, Z -4.6667, A 0.000, B 0.000, C 0.000 }
gfCNCPoint3[17499] = {X 80.3511, Y 46.1898, Z -4.6667, A 0.000, B 0.000, C 0.000 }
gfCNCPoint3[17500] = {X 80.1320, Y 47.3615, Z -4.6667, A 0.000, B 0.000, C 0.000 }
gfCNCPoint3[17501] = {X 79.7706, Y 48.4974, Z -4.6667, A 0.000, B 0.000, C 0.000 }
gfCNCPoint3[17502] = {X 79.2722, Y 49.5803, Z -4.6667, A 0.000, B 0.000, C 0.000 }
gfCNCPoint3[17503] = {X 78.4688, Y 50.8341, Z -4.6667, A 0.000, B 0.000, C 0.000 }
gfCNCPoint3[17504] = {X 77.4826, Y 51.9498, Z -4.6667, A 0.000, B 0.000, C 0.000 }
gfCNCPoint3[17505] = {X 76.3369, Y 52.9011, Z -4.6667, A 0.000, B 0.000, C 0.000 }
gfCNCPoint3[17506] = {X 75.0589, Y 53.6653, Z -4.6667, A 0.000, B 0.000, C 0.000 }
gfCNCPoint3[17507] = {X 73.6787, Y 54.2246, Z -4.6667, A 0.000, B 0.000, C 0.000 }
gfCNCPoint3[17508] = {X 72.2292, Y 54.5655, Z -4.6667, A 0.000, B 0.000, C 0.000 }
gfCNCPoint3[17509] = {X 70.7445, Y 54.6800, Z -4.6667, A 0.000, B 0.000, C 0.000 }
gfCNCPoint3[17510] = {X 64.1851, Y 54.6800, Z -4.6667, A 0.000, B 0.000, C 0.000 }
gfCNCPoint3[17511] = {X 62.7229, Y 54.5689, Z -4.6667, A 0.000, B 0.000, C 0.000 }
gfCNCPoint3[17512] = {X 61.2943, Y 54.2383, Z -4.6667, A 0.000, B 0.000, C 0.000 }
gfCNCPoint3[17513] = {X 59.9320, Y 53.6956, Z -4.6667, A 0.000, B 0.000, C 0.000 }
gfCNCPoint3[17514] = {X 58.6673, Y 52.9534, Z -4.6667, A 0.000, B 0.000, C 0.000 }
gfCNCPoint3[17515] = {X 57.5293, Y 52.0286, Z -4.6667, A 0.000, B 0.000, C 0.000 }
gfCNCPoint3[17516] = {X 56.6337, Y 51.0563, Z -4.6667, A 0.000, B 0.000, C 0.000 }
gfCNCPoint3[17517] = {X 55.8790, Y 49.9710, Z -4.6667, A 0.000, B 0.000, C 0.000 }
gfCNCPoint3[17518] = {X 55.1243, Y 51.0563, Z -4.6667, A 0.000, B 0.000, C 0.000 }
gfCNCPoint3[17519] = {X 54.2288, Y 52.0286, Z -4.6667, A 0.000, B 0.000, C 0.000 }
gfCNCPoint3[17520] = {X 53.0907, Y 52.9534, Z -4.6667, A 0.000, B 0.000, C 0.000 }
gfCNCPoint3[17521] = {X 51.8261, Y 53.6956, Z -4.6667, A 0.000, B 0.000, C 0.000 }
gfCNCPoint3[17522] = {X 50.4638, Y 54.2383, Z -4.6667, A 0.000, B 0.000, C 0.000 }
gfCNCPoint3[17523] = {X 49.0351, Y 54.5689, Z -4.6667, A 0.000, B 0.000, C 0.000 }
gfCNCPoint3[17524] = {X 47.5729, Y 54.6800, Z -4.6667, A 0.000, B 0.000, C 0.000 }
gfCNCPoint3[17525] = {X 40.6393, Y 54.6800, Z -4.6667, A 0.000, B 0.000, C 0.000 }
gfCNCPoint3[17526] = {X 39.2448, Y 54.5790, Z -4.6667, A 0.000, B 0.000, C 0.000 }
gfCNCPoint3[17527] = {X 37.8793, Y 54.2782, Z -4.6667, A 0.000, B 0.000, C 0.000 }
gfCNCPoint3[17528] = {X 36.5715, Y 53.7838, Z -4.6667, A 0.000, B 0.000, C 0.000 }
gfCNCPoint3[17529] = {X 35.3485, Y 53.1062, Z -4.6667, A 0.000, B 0.000, C 0.000 }
gfCNCPoint3[17530] = {X 33.9152, Y 54.1345, Z -4.6667, A 0.000, B 0.000, C 0.000 }
gfCNCPoint3[17531] = {X 32.3639, Y 54.9747, Z -4.6667, A 0.000, B 0.000, C 0.000 }
gfCNCPoint3[17532] = {X 30.7195, Y 55.6133, Z -4.6667, A 0.000, B 0.000, C 0.000 }
gfCNCPoint3[17533] = {X 29.0078, Y 56.0403, Z -4.6667, A 0.000, B 0.000, C 0.000 }
gfCNCPoint3[17534] = {X 27.2561, Y 56.2488, Z -4.6667, A 0.000, B 0.000, C 0.000 }
gfCNCPoint3[17535] = {X 24.9824, Y 57.2320, Z -4.6667, A 0.000, B 0.000, C 0.000 }
gfCNCPoint3[17536] = {X 22.6507, Y 58.0684, Z -4.6667, A 0.000, B 0.000, C 0.000 }
gfCNCPoint3[17537] = {X 20.0881, Y 58.7973, Z -4.6667, A 0.000, B 0.000, C 0.000 }
gfCNCPoint3[17538] = {X 17.4744, Y 59.3135, Z -4.6667, A 0.000, B 0.000, C 0.000 }
gfCNCPoint3[17539] = {X 14.8271, Y 59.6137, Z -4.6667, A 0.000, B 0.000, C 0.000 }
gfCNCPoint3[17540] = {X 12.1641, Y 59.6957, Z -4.6667, A 0.000, B 0.000, C 0.000 }
gfCNCPoint3[17541] = {X 9.5034, Y 59.5591, Z -4.6667, A 0.000, B 0.000, C 0.000 }
gfCNCPoint3[17542] = {X 9.5034, Y 90.4950, Z -4.6667, A 0.000, B 0.000, C 0.000 }
gfCNCPoint3[17543] = {X 114.8635, Y 90.4950, Z -4.6667, A 0.000, B 0.000, C 0.000 }
gfCNCPoint3[17544] = {X 115.7477, Y 89.2992, Z -4.6667, A 0.000, B 0.000, C 0.000 }
gfCNCPoint3[17545] = {X 116.7722, Y 88.2211, Z -4.6667, A 0.000, B 0.000, C 0.000 }
gfCNCPoint3[17546] = {X 117.9215, Y 87.2771, Z -4.6667, A 0.000, B 0.000, C 0.000 }
gfCNCPoint3[17547] = {X 119.1780, Y 86.4815, Z -4.6667, A 0.000, B 0.000, C 0.000 }
gfCNCPoint3[17548] = {X 120.5228, Y 85.8463, Z -4.6667, A 0.000, B 0.000, C 0.000 }
gfCNCPoint3[17549] = {X 121.9354, Y 85.3811, Z -4.6667, A 0.000, B 0.000, C 0.000 }
gfCNCPoint3[17550] = {X 123.3945, Y 85.0931, Z -4.6667, A 0.000, B 0.000, C 0.000 }
gfCNCPoint3[17551] = {X 123.5612, Y 84.9136, Z -4.6667, A 0.000, B 0.000, C 0.000 }
gfCNCPoint3[17552] = {X 123.7260, Y 84.7324, Z -4.6667, A 0.000, B 0.000, C 0.000 }
gfCNCPoint3[17553] = {X 147.2181, Y 58.9347, Z -4.6667, A 0.000, B 0.000, C 0.000 }
gfCNCPoint3[17554] = {X 147.2180, Y 58.0000, Z -4.6667, A 0.000, B 0.000, C 0.000 }
gfCNCPoint3[17555] = {X 147.2987, Y 56.6058, Z -4.6667, A 0.000, B 0.000, C 0.000 }
gfCNCPoint3[17556] = {X 147.5398, Y 55.2303, Z -4.6667, A 0.000, B 0.000, C 0.000 }
gfCNCPoint3[17557] = {X 148.0022, Y 53.7185, Z -4.6667, A 0.000, B 0.000, C 0.000 }
gfCNCPoint3[17558] = {X 148.6580, Y 52.2800, Z -4.6667, A 0.000, B 0.000, C 0.000 }
gfCNCPoint3[17559] = {X 143.0396, Y 52.2800, Z -4.6667, A 0.000, B 0.000, C 0.000 }
gfCNCPoint3[17560] = {X 141.7807, Y 52.1703, Z -4.6667, A 0.000, B 0.000, C 0.000 }
gfCNCPoint3[17561] = {X 140.5597, Y 51.8446, Z -4.6667, A 0.000, B 0.000, C 0.000 }
gfCNCPoint3[17562] = {X 139.4134, Y 51.3126, Z -4.6667, A 0.000, B 0.000, C 0.000 }
gfCNCPoint3[17563] = {X 138.3764, Y 50.5904, Z -4.6667, A 0.000, B 0.000, C 0.000 }
gfCNCPoint3[17564] = {X 137.4799, Y 49.6998, Z -4.6667, A 0.000, B 0.000, C 0.000 }
gfCNCPoint3[17565] = {X 136.7509, Y 48.6675, Z -4.6667, A 0.000, B 0.000, C 0.000 }
gfCNCPoint3[17566] = {X 136.2114, Y 47.5248, Z -4.6667, A 0.000, B 0.000, C 0.000 }
gfCNCPoint3[17567] = {X 135.8777, Y 46.3059, Z -4.6667, A 0.000, B 0.000, C 0.000 }
gfCNCPoint3[17568] = {X 135.7598, Y 45.0477, Z -4.6667, A 0.000, B 0.000, C 0.000 }
gfCNCPoint3[17569] = {X 135.7601, Y 44.1247, Z -4.6667, A 0.000, B 0.000, C 0.000 }
gfCNCPoint3[17570] = {X 135.8408, Y 43.1249, Z -4.6667, A 0.000, B 0.000, C 0.000 }
gfCNCPoint3[17571] = {X 136.0581, Y 42.1457, Z -4.6667, A 0.000, B 0.000, C 0.000 }
gfCNCPoint3[17572] = {X 138.3597, Y 42.8258, Z -4.6667, A 0.000, B 0.000, C 0.000 }
gfCNCPoint3[17573] = {X 138.6721, Y 42.0319, Z -4.6667, A 0.000, B 0.000, C 0.000 }
gfCNCPoint3[17574] = {X 139.1179, Y 41.3046, Z -4.6667, A 0.000, B 0.000, C 0.000 }
gfCNCPoint3[17575] = {X 139.6836, Y 40.6660, Z -4.6667, A 0.000, B 0.000, C 0.000 }
gfCNCPoint3[17576] = {X 139.6836, Y 20.4374, Z -4.6667, A 0.000, B 0.000, C 0.000 }
gfCNCPoint3[17577] = {X 137.7103, Y 20.4370, Z -4.6667, A 0.000, B 0.000, C 0.000 }
gfCNCPoint3[17578] = {X 137.0000, Y 21.1822, Z -4.6667, A 0.000, B 0.000, C 0.000 }
gfCNCPoint3[17579] = {X 136.1491, Y 21.7619, Z -4.6667, A 0.000, B 0.000, C 0.000 }
gfCNCPoint3[17580] = {X 135.4282, Y 22.0767, Z -4.6667, A 0.000, B 0.000, C 0.000 }
gfCNCPoint3[17581] = {X 134.6660, Y 22.2715, Z -4.6667, A 0.000, B 0.000, C 0.000 }
gfCNCPoint3[17582] = {X 133.8824, Y 22.3414, Z -4.6667, A 0.000, B 0.000, C 0.000 }
gfCNCPoint3[17583] = {X 133.2006, Y 22.3415, Z -4.6667, A 0.000, B 0.000, C 0.000 }
gfCNCPoint3[17584] = {X 132.2486, Y 22.2478, Z -4.6667, A 0.000, B 0.000, C 0.000 }
gfCNCPoint3[17585] = {X 131.3331, Y 21.9701, Z -4.6667, A 0.000, B 0.000, C 0.000 }
gfCNCPoint3[17586] = {X 130.4895, Y 21.5191, Z -4.6667, A 0.000, B 0.000, C 0.000 }
gfCNCPoint3[17587] = {X 129.7500, Y 20.9122, Z -4.6667, A 0.000, B 0.000, C 0.000 }
gfCNCPoint3[17588] = {X 129.1431, Y 20.1727, Z -4.6667, A 0.000, B 0.000, C 0.000 }
gfCNCPoint3[17589] = {X 128.6921, Y 19.3290, Z -4.6667, A 0.000, B 0.000, C 0.000 }
gfCNCPoint3[17590] = {X 128.4144, Y 18.4136, Z -4.6667, A 0.000, B 0.000, C 0.000 }
gfCNCPoint3[17591] = {X 128.3206, Y 17.4615, Z -4.6667, A 0.000, B 0.000, C 0.000 }
gfCNCPoint3[17592] = {X 128.3206, Y 10.4835, Z -4.6667, A 0.000, B 0.000, C 0.000 }
gfCNCPoint3[17593] = {X 128.3317, Y 10.1548, Z -4.6667, A 0.000, B 0.000, C 0.000 }
gfCNCPoint3[17594] = {X 128.3649, Y 9.8276, Z -4.6667, A 0.000, B 0.000, C 0.000 }
gfCNCPoint3[17595] = {X 128.6078, Y 8.8341, Z -4.6667, A 0.000, B 0.000, C 0.000 }
gfCNCPoint3[17596] = {X 129.0525, Y 7.9131, Z -4.6667, A 0.000, B 0.000, C 0.000 }
gfCNCPoint3[17597] = {X 129.6793, Y 7.1050, Z -4.6667, A 0.000, B 0.000, C 0.000 }
gfCNCPoint3[17598] = {X 130.0257, Y 7.4373, Z -4.6667, A 0.000, B 0.000, C 0.000 }
gfCNCPoint3[17599] = {X 130.6997, Y 6.8634, Z -4.6667, A 0.000, B 0.000, C 0.000 }
gfCNCPoint3[17600] = {X 131.4749, Y 6.4361, Z -4.6667, A 0.000, B 0.000, C 0.000 }
gfCNCPoint3[17601] = {X 132.3199, Y 6.1726, Z -4.6667, A 0.000, B 0.000, C 0.000 }
gfCNCPoint3[17602] = {X 133.2007, Y 6.0835, Z -4.6667, A 0.000, B 0.000, C 0.000 }
gfCNCPoint3[17603] = {X 133.8874, Y 6.0837, Z -4.6667, A 0.000, B 0.000, C 0.000 }
gfCNCPoint3[17604] = {X 134.7188, Y 6.1717, Z -4.6667, A 0.000, B 0.000, C 0.000 }
gfCNCPoint3[17605] = {X 135.5186, Y 6.4153, Z -4.6667, A 0.000, B 0.000, C 0.000 }
gfCNCPoint3[17606] = {X 136.2579, Y 6.8059, Z -4.6667, A 0.000, B 0.000, C 0.000 }
gfCNCPoint3[17607] = {X 136.9099, Y 7.3292, Z -4.6667, A 0.000, B 0.000, C 0.000 }
gfCNCPoint3[17608] = {X 137.4512, Y 7.9664, Z -4.6667, A 0.000, B 0.000, C 0.000 }
gfCNCPoint3[17609] = {X 155.0716, Y 7.9664, Z -4.6667, A 0.000, B 0.000, C 0.000 }
gfCNCPoint3[17610] = {X 155.6193, Y 7.3229, Z -4.6667, A 0.000, B 0.000, C 0.000 }
gfCNCPoint3[17611] = {X 156.2800, Y 6.7960, Z -4.6667, A 0.000, B 0.000, C 0.000 }
gfCNCPoint3[17612] = {X 157.0293, Y 6.4051, Z -4.6667, A 0.000, B 0.000, C 0.000 }
gfCNCPoint3[17613] = {X 157.8394, Y 6.1646, Z -4.6667, A 0.000, B 0.000, C 0.000 }
gfCNCPoint3[17614] = {X 158.6806, Y 6.0835, Z -4.6667, A 0.000, B 0.000, C 0.000 }
gfCNCPoint3[17615] = {X 159.3791, Y 6.0839, Z -4.6667, A 0.000, B 0.000, C 0.000 }
gfCNCPoint3[17616] = {X 160.3488, Y 6.2050, Z -4.6667, A 0.000, B 0.000, C 0.000 }
gfCNCPoint3[17617] = {X 161.2678, Y 6.5371, Z -4.6667, A 0.000, B 0.000, C 0.000 }
gfCNCPoint3[17618] = {X 162.0908, Y 7.0639, Z -4.6667, A 0.000, B 0.000, C 0.000 }
gfCNCPoint3[17619] = {X 162.7773, Y 7.7593, Z -4.6667, A 0.000, B 0.000, C 0.000 }
gfCNCPoint3[17620] = {X 163.2934, Y 8.5891, Z -4.6667, A 0.000, B 0.000, C 0.000 }
gfCNCPoint3[17621] = {X 163.6136, Y 9.5124, Z -4.6667, A 0.000, B 0.000, C 0.000 }
gfCNCPoint3[17622] = {X 163.7221, Y 10.4835, Z -4.6667, A 0.000, B 0.000, C 0.000 }
gfCNCPoint3[17623] = {X 163.7221, Y 17.4615, Z -4.6667, A 0.000, B 0.000, C 0.000 }
gfCNCPoint3[17624] = {X 163.6118, Y 18.4406, Z -4.6667, A 0.000, B 0.000, C 0.000 }
gfCNCPoint3[17625] = {X 163.2863, Y 19.3706, Z -4.6667, A 0.000, B 0.000, C 0.000 }
gfCNCPoint3[17626] = {X 162.7621, Y 20.2049, Z -4.6667, A 0.000, B 0.000, C 0.000 }
gfCNCPoint3[17627] = {X 162.0654, Y 20.9016, Z -4.6667, A 0.000, B 0.000, C 0.000 }
gfCNCPoint3[17628] = {X 161.2312, Y 21.4258, Z -4.6667, A 0.000, B 0.000, C 0.000 }
gfCNCPoint3[17629] = {X 160.3012, Y 21.7512, Z -4.6667, A 0.000, B 0.000, C 0.000 }
gfCNCPoint3[17630] = {X 159.3221, Y 21.8615, Z -4.6667, A 0.000, B 0.000, C 0.000 }
gfCNCPoint3[17631] = {X 158.6789, Y 21.8615, Z -4.6667, A 0.000, B 0.000, C 0.000 }
gfCNCPoint3[17632] = {X 157.8334, Y 21.7766, Z -4.6667, A 0.000, B 0.000, C 0.000 }
gfCNCPoint3[17633] = {X 157.0197, Y 21.5320, Z -4.6667, A 0.000, B 0.000, C 0.000 }
gfCNCPoint3[17634] = {X 156.2676, Y 21.1367, Z -4.6667, A 0.000, B 0.000, C 0.000 }
gfCNCPoint3[17635] = {X 155.6047, Y 20.6051, Z -4.6667, A 0.000, B 0.000, C 0.000 }
gfCNCPoint3[17636] = {X 155.0553, Y 19.9570, Z -4.6667, A 0.000, B 0.000, C 0.000 }
gfCNCPoint3[17637] = {X 152.3565, Y 19.9581, Z -4.6667, A 0.000, B 0.000, C 0.000 }
gfCNCPoint3[17638] = {X 152.3551, Y 40.8428, Z -4.6667, A 0.000, B 0.000, C 0.000 }
gfCNCPoint3[17639] = {X 152.8074, Y 41.3304, Z -4.6667, A 0.000, B 0.000, C 0.000 }
gfCNCPoint3[17640] = {X 152.9000, Y 41.4410, Z -4.6667, A 0.000, B 0.000, C 0.000 }
gfCNCPoint3[17641] = {X 153.4344, Y 42.2813, Z -4.6667, A 0.000, B 0.000, C 0.000 }
gfCNCPoint3[17642] = {X 153.7677, Y 43.2197, Z -4.6667, A 0.000, B 0.000, C 0.000 }
gfCNCPoint3[17643] = {X 153.8831, Y 44.2089, Z -4.6667, A 0.000, B 0.000, C 0.000 }
gfCNCPoint3[17644] = {X 153.8829, Y 45.0423, Z -4.6667, A 0.000, B 0.000, C 0.000 }
gfCNCPoint3[17645] = {X 153.7646, Y 46.0144, Z -4.6667, A 0.000, B 0.000, C 0.000 }
gfCNCPoint3[17646] = {X 153.4342, Y 46.9363, Z -4.6667, A 0.000, B 0.000, C 0.000 }
gfCNCPoint3[17647] = {X 152.9080, Y 47.7622, Z -4.6667, A 0.000, B 0.000, C 0.000 }
gfCNCPoint3[17648] = {X 152.2123, Y 48.4513, Z -4.6667, A 0.000, B 0.000, C 0.000 }
gfCNCPoint3[17649] = {X 151.3813, Y 48.9695, Z -4.6667, A 0.000, B 0.000, C 0.000 }
gfCNCPoint3[17650] = {X 150.4563, Y 49.2910, Z -4.6667, A 0.000, B 0.000, C 0.000 }
gfCNCPoint3[17651] = {X 149.4831, Y 49.4000, Z -4.6667, A 0.000, B 0.000, C 0.000 }
gfCNCPoint3[17652] = {X 143.0396, Y 49.4000, Z -4.6667, A 0.000, B 0.000, C 0.000 }
gfCNCPoint3[17653] = {X 142.0605, Y 49.2897, Z -4.6667, A 0.000, B 0.000, C 0.000 }
gfCNCPoint3[17654] = {X 141.1305, Y 48.9643, Z -4.6667, A 0.000, B 0.000, C 0.000 }
gfCNCPoint3[17655] = {X 140.2963, Y 48.4400, Z -4.6667, A 0.000, B 0.000, C 0.000 }
gfCNCPoint3[17656] = {X 139.5996, Y 47.7433, Z -4.6667, A 0.000, B 0.000, C 0.000 }
gfCNCPoint3[17657] = {X 139.0754, Y 46.9091, Z -4.6667, A 0.000, B 0.000, C 0.000 }
gfCNCPoint3[17658] = {X 138.7499, Y 45.9791, Z -4.6667, A 0.000, B 0.000, C 0.000 }
gfCNCPoint3[17659] = {X 138.6396, Y 45.0000, Z -4.6667, A 0.000, B 0.000, C 0.000 }
gfCNCPoint3[17660] = {X 138.6400, Y 44.1483, Z -4.6667, A 0.000, B 0.000, C 0.000 }
gfCNCPoint3[17661] = {X 138.7505, Y 43.2275, Z -4.6667, A 0.000, B 0.000, C 0.000 }
gfCNCPoint3[17662] = {X 139.0514, Y 42.3503, Z -4.6667, A 0.000, B 0.000, C 0.000 }
gfCNCPoint3[17663] = {X 139.5295, Y 41.5556, Z -4.6667, A 0.000, B 0.000, C 0.000 }
gfCNCPoint3[17664] = {X 140.1636, Y 40.8789, Z -4.6667, A 0.000, B 0.000, C 0.000 }
gfCNCPoint3[17665] = {X 140.1636, Y 19.9575, Z -4.6667, A 0.000, B 0.000, C 0.000 }
gfCNCPoint3[17666] = {X 137.4663, Y 19.9569, Z -4.6667, A 0.000, B 0.000, C 0.000 }
gfCNCPoint3[17667] = {X 136.9186, Y 20.6074, Z -4.6667, A 0.000, B 0.000, C 0.000 }
gfCNCPoint3[17668] = {X 136.2560, Y 21.1404, Z -4.6667, A 0.000, B 0.000, C 0.000 }
gfCNCPoint3[17669] = {X 135.5033, Y 21.5360, Z -4.6667, A 0.000, B 0.000, C 0.000 }
gfCNCPoint3[17670] = {X 134.6885, Y 21.7794, Z -4.6667, A 0.000, B 0.000, C 0.000 }
gfCNCPoint3[17671] = {X 133.8422, Y 21.8615, Z -4.6667, A 0.000, B 0.000, C 0.000 }
gfCNCPoint3[17672] = {X 133.2006, Y 21.8615, Z -4.6667, A 0.000, B 0.000, C 0.000 }
gfCNCPoint3[17673] = {X 132.2215, Y 21.7512, Z -4.6667, A 0.000, B 0.000, C 0.000 }
gfCNCPoint3[17674] = {X 131.2916, Y 21.4258, Z -4.6667, A 0.000, B 0.000, C 0.000 }
gfCNCPoint3[17675] = {X 130.4573, Y 20.9016, Z -4.6667, A 0.000, B 0.000, C 0.000 }
gfCNCPoint3[17676] = {X 129.7606, Y 20.2049, Z -4.6667, A 0.000, B 0.000, C 0.000 }
gfCNCPoint3[17677] = {X 129.2364, Y 19.3706, Z -4.6667, A 0.000, B 0.000, C 0.000 }
gfCNCPoint3[17678] = {X 128.9110, Y 18.4406, Z -4.6667, A 0.000, B 0.000, C 0.000 }
gfCNCPoint3[17679] = {X 128.8006, Y 17.4615, Z -4.6667, A 0.000, B 0.000, C 0.000 }
gfCNCPoint3[17680] = {X 128.8006, Y 10.4835, Z -4.6667, A 0.000, B 0.000, C 0.000 }
gfCNCPoint3[17681] = {X 128.8808, Y 9.6475, Z -4.6667, A 0.000, B 0.000, C 0.000 }
gfCNCPoint3[17682] = {X 129.1184, Y 8.8419, Z -4.6667, A 0.000, B 0.000, C 0.000 }
gfCNCPoint3[17683] = {X 129.5047, Y 8.0961, Z -4.6667, A 0.000, B 0.000, C 0.000 }
gfCNCPoint3[17684] = {X 130.0257, Y 7.4373, Z -4.6667, A 0.000, B 0.000, C 0.000 }
gfCNCPoint3[17685] = {X 129.6793, Y 7.1050, Z -4.6667, A 0.000, B 0.000, C 0.000 }
gfCNCPoint3[17686] = {X 102.4337, Y 7.1050, Z -4.6667, A 0.000, B 0.000, C 0.000 }
gfCNCPoint3[17687] = {X 102.4337, Y 11.9050, Z -4.6667, A 0.000, B 0.000, C 0.000 }
gfCNCPoint3[17688] = {X 101.3242, Y 11.9050, Z -4.6667, A 0.000, B 0.000, C 0.000 }
gfCNCPoint3[17689] = {X 101.3283, Y 12.0459, Z -4.6667, A 0.000, B 0.000, C 0.000 }
gfCNCPoint3[17690] = {X 101.3297, Y 12.1868, Z -4.6667, A 0.000, B 0.000, C 0.000 }
gfCNCPoint3[17691] = {X 101.3293, Y 13.0462, Z -4.6667, A 0.000, B 0.000, C 0.000 }
gfCNCPoint3[17692] = {X 101.2275, Y 14.1936, Z -4.6667, A 0.000, B 0.000, C 0.000 }
gfCNCPoint3[17693] = {X 100.9458, Y 15.3107, Z -4.6667, A 0.000, B 0.000, C 0.000 }
gfCNCPoint3[17694] = {X 101.0397, Y 15.5443, Z -4.6667, A 0.000, B 0.000, C 0.000 }
gfCNCPoint3[17695] = {X 101.8684, Y 17.5986, Z -4.6667, A 0.000, B 0.000, C 0.000 }
gfCNCPoint3[17696] = {X 102.8002, Y 15.2750, Z -4.6667, A 0.000, B 0.000, C 0.000 }
gfCNCPoint3[17697] = {X 102.5273, Y 14.1747, Z -4.6667, A 0.000, B 0.000, C 0.000 }
gfCNCPoint3[17698] = {X 102.4286, Y 13.0453, Z -4.6667, A 0.000, B 0.000, C 0.000 }
gfCNCPoint3[17699] = {X 102.4283, Y 12.1868, Z -4.6667, A 0.000, B 0.000, C 0.000 }
gfCNCPoint3[17700] = {X 102.4296, Y 12.0459, Z -4.6667, A 0.000, B 0.000, C 0.000 }
gfCNCPoint3[17701] = {X 102.4337, Y 11.9050, Z -4.6667, A 0.000, B 0.000, C 0.000 }
gfCNCPoint3[17702] = {X 102.4337, Y 9.5050, Z -4.6667, A 0.000, B 0.000, C 0.000 }
gfCNCPoint3[17703] = {X 98.1267, Y 9.5050, Z -4.6667, A 0.000, B 0.000, C 0.000 }
gfCNCPoint3[17704] = {X 98.5429, Y 10.2829, Z -4.6667, A 0.000, B 0.000, C 0.000 }
gfCNCPoint3[17705] = {X 98.8123, Y 11.1230, Z -4.6667, A 0.000, B 0.000, C 0.000 }
gfCNCPoint3[17706] = {X 98.9260, Y 11.9979, Z -4.6667, A 0.000, B 0.000, C 0.000 }
gfCNCPoint3[17707] = {X 98.9288, Y 12.0923, Z -4.6667, A 0.000, B 0.000, C 0.000 }
gfCNCPoint3[17708] = {X 98.9297, Y 12.1868, Z -4.6667, A 0.000, B 0.000, C 0.000 }
gfCNCPoint3[17709] = {X 98.9294, Y 13.0237, Z -4.6667, A 0.000, B 0.000, C 0.000 }
gfCNCPoint3[17710] = {X 98.8590, Y 13.8057, Z -4.6667, A 0.000, B 0.000, C 0.000 }
gfCNCPoint3[17711] = {X 98.6639, Y 14.5664, Z -4.6667, A 0.000, B 0.000, C 0.000 }
gfCNCPoint3[17712] = {X 98.3495, Y 15.2858, Z -4.6667, A 0.000, B 0.000, C 0.000 }
gfCNCPoint3[17713] = {X 98.8133, Y 16.4405, Z -4.6667, A 0.000, B 0.000, C 0.000 }
gfCNCPoint3[17714] = {X 101.8752, Y 24.0304, Z -4.6667, A 0.000, B 0.000, C 0.000 }
gfCNCPoint3[17715] = {X 105.3931, Y 15.2570, Z -4.6667, A 0.000, B 0.000, C 0.000 }
gfCNCPoint3[17716] = {X 105.0869, Y 14.5456, Z -4.6667, A 0.000, B 0.000, C 0.000 }
gfCNCPoint3[17717] = {X 104.8971, Y 13.7946, Z -4.6667, A 0.000, B 0.000, C 0.000 }
gfCNCPoint3[17718] = {X 104.8285, Y 13.0231, Z -4.6667, A 0.000, B 0.000, C 0.000 }
gfCNCPoint3[17719] = {X 104.8283, Y 12.1868, Z -4.6667, A 0.000, B 0.000, C 0.000 }
gfCNCPoint3[17720] = {X 104.8292, Y 12.0923, Z -4.6667, A 0.000, B 0.000, C 0.000 }
gfCNCPoint3[17721] = {X 104.8319, Y 11.9979, Z -4.6667, A 0.000, B 0.000, C 0.000 }
gfCNCPoint3[17722] = {X 104.9456, Y 11.1230, Z -4.6667, A 0.000, B 0.000, C 0.000 }
gfCNCPoint3[17723] = {X 105.2150, Y 10.2829, Z -4.6667, A 0.000, B 0.000, C 0.000 }
gfCNCPoint3[17724] = {X 105.6313, Y 9.5050, Z -4.6667, A 0.000, B 0.000, C 0.000 }
gfCNCPoint3[17725] = {X 102.4337, Y 9.5050, Z -4.6667, A 0.000, B 0.000, C 0.000 }
gfCNCPoint3[17726] = {X 102.4337, Y 7.1050, Z -4.6667, A 0.000, B 0.000, C 0.000 }
gfCNCPoint3[17727] = {X 64.8349, Y 7.1050, Z -4.6667, A 0.000, B 0.000, C 0.000 }
gfCNCPoint3[17728] = {X 65.5946, Y 8.0241, Z -4.6667, A 0.000, B 0.000, C 0.000 }
gfCNCPoint3[17729] = {X 66.1940, Y 9.0550, Z -4.6667, A 0.000, B 0.000, C 0.000 }
gfCNCPoint3[17730] = {X 66.6172, Y 10.1699, Z -4.6667, A 0.000, B 0.000, C 0.000 }
gfCNCPoint3[17731] = {X 66.8305, Y 11.1683, Z -4.6667, A 0.000, B 0.000, C 0.000 }
gfCNCPoint3[17732] = {X 66.9021, Y 12.1868, Z -4.6667, A 0.000, B 0.000, C 0.000 }
gfCNCPoint3[17733] = {X 66.9018, Y 13.0462, Z -4.6667, A 0.000, B 0.000, C 0.000 }
gfCNCPoint3[17734] = {X 66.7772, Y 14.3208, Z -4.6667, A 0.000, B 0.000, C 0.000 }
gfCNCPoint3[17735] = {X 66.4312, Y 15.5539, Z -4.6667, A 0.000, B 0.000, C 0.000 }
gfCNCPoint3[17736] = {X 74.9117, Y 38.2395, Z -4.6667, A 0.000, B 0.000, C 0.000 }
gfCNCPoint3[17737] = {X 75.8039, Y 38.9743, Z -4.6667, A 0.000, B 0.000, C 0.000 }
gfCNCPoint3[17738] = {X 76.5686, Y 39.8410, Z -4.6667, A 0.000, B 0.000, C 0.000 }
gfCNCPoint3[17739] = {X 77.1865, Y 40.8179, Z -4.6667, A 0.000, B 0.000, C 0.000 }
gfCNCPoint3[17740] = {X 77.6420, Y 41.8802, Z -4.6667, A 0.000, B 0.000, C 0.000 }
gfCNCPoint3[17741] = {X 77.9236, Y 43.0012, Z -4.6667, A 0.000, B 0.000, C 0.000 }
gfCNCPoint3[17742] = {X 78.0243, Y 44.1527, Z -4.6667, A 0.000, B 0.000, C 0.000 }
gfCNCPoint3[17743] = {X 78.0245, Y 45.0000, Z -4.6667, A 0.000, B 0.000, C 0.000 }
gfCNCPoint3[17744] = {X 77.9139, Y 46.2642, Z -4.6667, A 0.000, B 0.000, C 0.000 }
gfCNCPoint3[17745] = {X 77.5854, Y 47.4899, Z -4.6667, A 0.000, B 0.000, C 0.000 }
gfCNCPoint3[17746] = {X 77.0491, Y 48.6400, Z -4.6667, A 0.000, B 0.000, C 0.000 }
gfCNCPoint3[17747] = {X 76.3213, Y 49.6795, Z -4.6667, A 0.000, B 0.000, C 0.000 }
gfCNCPoint3[17748] = {X 75.4240, Y 50.5768, Z -4.6667, A 0.000, B 0.000, C 0.000 }
gfCNCPoint3[17749] = {X 74.3845, Y 51.3047, Z -4.6667, A 0.000, B 0.000, C 0.000 }
gfCNCPoint3[17750] = {X 73.2344, Y 51.8410, Z -4.6667, A 0.000, B 0.000, C 0.000 }
gfCNCPoint3[17751] = {X 72.0086, Y 52.1694, Z -4.6667, A 0.000, B 0.000, C 0.000 }
gfCNCPoint3[17752] = {X 70.7445, Y 52.2800, Z -4.6667, A 0.000, B 0.000, C 0.000 }
gfCNCPoint3[17753] = {X 64.1851, Y 52.2800, Z -4.6667, A 0.000, B 0.000, C 0.000 }
gfCNCPoint3[17754] = {X 62.9397, Y 52.1727, Z -4.6667, A 0.000, B 0.000, C 0.000 }
gfCNCPoint3[17755] = {X 61.7311, Y 51.8539, Z -4.6667, A 0.000, B 0.000, C 0.000 }
gfCNCPoint3[17756] = {X 60.5947, Y 51.3330, Z -4.6667, A 0.000, B 0.000, C 0.000 }
gfCNCPoint3[17757] = {X 59.5643, Y 50.6255, Z -4.6667, A 0.000, B 0.000, C 0.000 }
gfCNCPoint3[17758] = {X 58.6700, Y 49.7521, Z -4.6667, A 0.000, B 0.000, C 0.000 }
gfCNCPoint3[17759] = {X 57.9384, Y 48.7385, Z -4.6667, A 0.000, B 0.000, C 0.000 }
gfCNCPoint3[17760] = {X 57.3706, Y 47.5614, Z -4.6667, A 0.000, B 0.000, C 0.000 }
gfCNCPoint3[17761] = {X 57.0224, Y 46.3017, Z -4.6667, A 0.000, B 0.000, C 0.000 }
gfCNCPoint3[17762] = {X 56.9051, Y 45.0000, Z -4.6667, A 0.000, B 0.000, C 0.000 }
gfCNCPoint3[17763] = {X 56.9051, Y 44.2048, Z -4.6667, A 0.000, B 0.000, C 0.000 }
gfCNCPoint3[17764] = {X 56.9286, Y 43.6252, Z -4.6667, A 0.000, B 0.000, C 0.000 }
gfCNCPoint3[17765] = {X 56.9981, Y 43.0492, Z -4.6667, A 0.000, B 0.000, C 0.000 }
gfCNCPoint3[17766] = {X 54.7600, Y 43.0492, Z -4.6667, A 0.000, B 0.000, C 0.000 }
gfCNCPoint3[17767] = {X 54.8275, Y 43.6012, Z -4.6667, A 0.000, B 0.000, C 0.000 }
gfCNCPoint3[17768] = {X 54.8528, Y 44.1567, Z -4.6667, A 0.000, B 0.000, C 0.000 }
gfCNCPoint3[17769] = {X 54.8529, Y 45.0000, Z -4.6667, A 0.000, B 0.000, C 0.000 }
gfCNCPoint3[17770] = {X 54.7356, Y 46.3017, Z -4.6667, A 0.000, B 0.000, C 0.000 }
gfCNCPoint3[17771] = {X 54.3875, Y 47.5614, Z -4.6667, A 0.000, B 0.000, C 0.000 }
gfCNCPoint3[17772] = {X 53.8197, Y 48.7385, Z -4.6667, A 0.000, B 0.000, C 0.000 }
gfCNCPoint3[17773] = {X 53.0880, Y 49.7521, Z -4.6667, A 0.000, B 0.000, C 0.000 }
gfCNCPoint3[17774] = {X 52.1938, Y 50.6255, Z -4.6667, A 0.000, B 0.000, C 0.000 }
gfCNCPoint3[17775] = {X 51.1633, Y 51.3330, Z -4.6667, A 0.000, B 0.000, C 0.000 }
gfCNCPoint3[17776] = {X 50.0270, Y 51.8539, Z -4.6667, A 0.000, B 0.000, C 0.000 }
gfCNCPoint3[17777] = {X 48.8183, Y 52.1727, Z -4.6667, A 0.000, B 0.000, C 0.000 }
gfCNCPoint3[17778] = {X 47.5729, Y 52.2800, Z -4.6667, A 0.000, B 0.000, C 0.000 }
gfCNCPoint3[17779] = {X 40.6393, Y 52.2800, Z -4.6667, A 0.000, B 0.000, C 0.000 }
gfCNCPoint3[17780] = {X 39.4476, Y 52.1818, Z -4.6667, A 0.000, B 0.000, C 0.000 }
gfCNCPoint3[17781] = {X 38.2881, Y 51.8899, Z -4.6667, A 0.000, B 0.000, C 0.000 }
gfCNCPoint3[17782] = {X 37.1919, Y 51.4120, Z -4.6667, A 0.000, B 0.000, C 0.000 }
gfCNCPoint3[17783] = {X 36.1888, Y 50.7612, Z -4.6667, A 0.000, B 0.000, C 0.000 }
gfCNCPoint3[17784] = {X 35.3058, Y 49.9550, Z -4.6667, A 0.000, B 0.000, C 0.000 }
gfCNCPoint3[17785] = {X 34.8234, Y 50.4196, Z -4.6667, A 0.000, B 0.000, C 0.000 }
gfCNCPoint3[17786] = {X 34.3150, Y 50.8555, Z -4.6667, A 0.000, B 0.000, C 0.000 }
gfCNCPoint3[17787] = {X 33.7759, Y 51.2914, Z -4.6667, A 0.000, B 0.000, C 0.000 }
gfCNCPoint3[17788] = {X 32.5173, Y 52.1768, Z -4.6667, A 0.000, B 0.000, C 0.000 }
gfCNCPoint3[17789] = {X 31.1528, Y 52.8882, Z -4.6667, A 0.000, B 0.000, C 0.000 }
gfCNCPoint3[17790] = {X 29.7062, Y 53.4128, Z -4.6667, A 0.000, B 0.000, C 0.000 }
gfCNCPoint3[17791] = {X 28.2029, Y 53.7416, Z -4.6667, A 0.000, B 0.000, C 0.000 }
gfCNCPoint3[17792] = {X 26.6693, Y 53.8688, Z -4.6667, A 0.000, B 0.000, C 0.000 }
gfCNCPoint3[17793] = {X 24.3216, Y 54.9117, Z -4.6667, A 0.000, B 0.000, C 0.000 }
gfCNCPoint3[17794] = {X 21.9063, Y 55.7868, Z -4.6667, A 0.000, B 0.000, C 0.000 }
gfCNCPoint3[17795] = {X 19.5320, Y 56.4626, Z -4.6667, A 0.000, B 0.000, C 0.000 }
gfCNCPoint3[17796] = {X 17.1103, Y 56.9413, Z -4.6667, A 0.000, B 0.000, C 0.000 }
gfCNCPoint3[17797] = {X 14.6575, Y 57.2197, Z -4.6667, A 0.000, B 0.000, C 0.000 }
gfCNCPoint3[17798] = {X 12.1901, Y 57.2958, Z -4.6667, A 0.000, B 0.000, C 0.000 }
gfCNCPoint3[17799] = {X 9.7248, Y 57.1693, Z -4.6667, A 0.000, B 0.000, C 0.000 }
gfCNCPoint3[17800] = {X 8.4101, Y 57.0183, Z -4.6667, A 0.000, B 0.000, C 0.000 }
gfCNCPoint3[17801] = {X 7.1034, Y 56.8096, Z -4.6667, A 0.000, B 0.000, C 0.000 }
gfCNCPoint3[17802] = {X 7.1034, Y 92.8950, Z -4.6667, A 0.000, B 0.000, C 0.000 }
gfCNCPoint3[17803] = {X 116.2647, Y 92.8950, Z -4.6667, A 0.000, B 0.000, C 0.000 }
gfCNCPoint3[17804] = {X 116.9717, Y 91.6577, Z -4.6667, A 0.000, B 0.000, C 0.000 }
gfCNCPoint3[17805] = {X 117.8528, Y 90.5376, Z -4.6667, A 0.000, B 0.000, C 0.000 }
gfCNCPoint3[17806] = {X 118.8888, Y 89.5589, Z -4.6667, A 0.000, B 0.000, C 0.000 }
gfCNCPoint3[17807] = {X 120.0572, Y 88.7430, Z -4.6667, A 0.000, B 0.000, C 0.000 }
gfCNCPoint3[17808] = {X 121.3327, Y 88.1075, Z -4.6667, A 0.000, B 0.000, C 0.000 }
gfCNCPoint3[17809] = {X 122.6878, Y 87.6661, Z -4.6667, A 0.000, B 0.000, C 0.000 }
gfCNCPoint3[17810] = {X 124.0930, Y 87.4285, Z -4.6667, A 0.000, B 0.000, C 0.000 }
gfCNCPoint3[17811] = {X 124.5363, Y 87.3616, Z -4.6667, A 0.000, B 0.000, C 0.000 }
gfCNCPoint3[17812] = {X 125.0278, Y 86.8591, Z -4.6667, A 0.000, B 0.000, C 0.000 }
gfCNCPoint3[17813] = {X 125.5051, Y 86.3432, Z -4.6667, A 0.000, B 0.000, C 0.000 }
gfCNCPoint3[17814] = {X 149.6585, Y 59.8193, Z -4.6667, A 0.000, B 0.000, C 0.000 }
gfCNCPoint3[17815] = {X 149.6295, Y 59.4066, Z -4.6667, A 0.000, B 0.000, C 0.000 }
gfCNCPoint3[17816] = {X 149.6181, Y 58.9930, Z -4.6667, A 0.000, B 0.000, C 0.000 }
gfCNCPoint3[17817] = {X 149.6180, Y 58.0000, Z -4.6667, A 0.000, B 0.000, C 0.000 }
gfCNCPoint3[17818] = {X 149.6915, Y 56.8093, Z -4.6667, A 0.000, B 0.000, C 0.000 }
gfCNCPoint3[17819] = {X 149.9109, Y 55.6367, Z -4.6667, A 0.000, B 0.000, C 0.000 }
gfCNCPoint3[17820] = {X 150.2729, Y 54.5000, Z -4.6667, A 0.000, B 0.000, C 0.000 }
gfCNCPoint3[17821] = {X 150.7719, Y 53.4164, Z -4.6667, A 0.000, B 0.000, C 0.000 }
gfCNCPoint3[17822] = {X 151.5117, Y 52.2488, Z -4.6667, A 0.000, B 0.000, C 0.000 }
gfCNCPoint3[17823] = {X 152.4103, Y 51.1984, Z -4.6667, A 0.000, B 0.000, C 0.000 }
gfCNCPoint3[17824] = {X 153.4493, Y 50.2867, Z -4.6667, A 0.000, B 0.000, C 0.000 }
gfCNCPoint3[17825] = {X 154.6075, Y 49.5323, Z -4.6667, A 0.000, B 0.000, C 0.000 }
gfCNCPoint3[17826] = {X 155.8614, Y 48.9505, Z -4.6667, A 0.000, B 0.000, C 0.000 }
gfCNCPoint3[17827] = {X 157.1854, Y 48.5533, Z -4.6667, A 0.000, B 0.000, C 0.000 }
gfCNCPoint3[17828] = {X 158.2353, Y 48.3785, Z -4.6667, A 0.000, B 0.000, C 0.000 }
gfCNCPoint3[17829] = {X 159.2980, Y 48.3200, Z -4.6667, A 0.000, B 0.000, C 0.000 }
gfCNCPoint3[17830] = {X 176.3097, Y 48.3200, Z -4.6667, A 0.000, B 0.000, C 0.000 }
gfCNCPoint3[17831] = {X 175.1957, Y 47.6609, Z -4.6667, A 0.000, B 0.000, C 0.000 }
gfCNCPoint3[17832] = {X 174.1331, Y 46.9217, Z -4.6667, A 0.000, B 0.000, C 0.000 }
gfCNCPoint3[17833] = {X 172.7671, Y 45.7590, Z -4.6667, A 0.000, B 0.000, C 0.000 }
gfCNCPoint3[17834] = {X 171.5635, Y 44.4288, Z -4.6667, A 0.000, B 0.000, C 0.000 }
gfCNCPoint3[17835] = {X 170.6255, Y 43.0901, Z -4.6667, A 0.000, B 0.000, C 0.000 }
gfCNCPoint3[17836] = {X 169.8525, Y 41.6499, Z -4.6667, A 0.000, B 0.000, C 0.000 }
gfCNCPoint3[17837] = {X 169.2552, Y 40.1283, Z -4.6667, A 0.000, B 0.000, C 0.000 }
gfCNCPoint3[17838] = {X 168.8421, Y 38.5468, Z -4.6667, A 0.000, B 0.000, C 0.000 }
gfCNCPoint3[17839] = {X 168.6189, Y 36.9275, Z -4.6667, A 0.000, B 0.000, C 0.000 }
gfCNCPoint3[17840] = {X 168.5329, Y 35.0258, Z -4.6667, A 0.000, B 0.000, C 0.000 }
gfCNCPoint3[17841] = {X 168.6852, Y 33.1282, Z -4.6667, A 0.000, B 0.000, C 0.000 }
gfCNCPoint3[17842] = {X 169.0735, Y 31.2646, Z -4.6667, A 0.000, B 0.000, C 0.000 }
gfCNCPoint3[17843] = {X 169.6918, Y 29.4641, Z -4.6667, A 0.000, B 0.000, C 0.000 }
gfCNCPoint3[17844] = {X 170.2638, Y 28.2674, Z -4.6667, A 0.000, B 0.000, C 0.000 }
gfCNCPoint3[17845] = {X 170.9707, Y 27.1451, Z -4.6667, A 0.000, B 0.000, C 0.000 }
gfCNCPoint3[17846] = {X 171.8029, Y 26.1124, Z -4.6667, A 0.000, B 0.000, C 0.000 }
gfCNCPoint3[17847] = {X 172.7493, Y 25.1831, Z -4.6667, A 0.000, B 0.000, C 0.000 }
gfCNCPoint3[17848] = {X 173.7971, Y 24.3699, Z -4.6667, A 0.000, B 0.000, C 0.000 }
gfCNCPoint3[17849] = {X 173.0270, Y 23.7517, Z -4.6667, A 0.000, B 0.000, C 0.000 }
gfCNCPoint3[17850] = {X 172.3971, Y 22.9911, Z -4.6667, A 0.000, B 0.000, C 0.000 }
gfCNCPoint3[17851] = {X 171.9332, Y 22.1192, Z -4.6667, A 0.000, B 0.000, C 0.000 }
gfCNCPoint3[17852] = {X 169.3220, Y 15.7237, Z -4.6667, A 0.000, B 0.000, C 0.000 }
gfCNCPoint3[17853] = {X 169.1088, Y 15.0753, Z -4.6667, A 0.000, B 0.000, C 0.000 }
gfCNCPoint3[17854] = {X 168.9882, Y 14.4035, Z -4.6667, A 0.000, B 0.000, C 0.000 }
gfCNCPoint3[17855] = {X 168.9599, Y 13.8791, Z -4.6667, A 0.000, B 0.000, C 0.000 }
gfCNCPoint3[17856] = {X 168.9882, Y 13.3548, Z -4.6667, A 0.000, B 0.000, C 0.000 }
gfCNCPoint3[17857] = {X 169.1590, Y 12.4995, Z -4.6667, A 0.000, B 0.000, C 0.000 }
gfCNCPoint3[17858] = {X 169.4794, Y 11.6882, Z -4.6667, A 0.000, B 0.000, C 0.000 }
gfCNCPoint3[17859] = {X 169.9390, Y 10.9470, Z -4.6667, A 0.000, B 0.000, C 0.000 }
gfCNCPoint3[17860] = {X 170.6135, Y 10.2179, Z -4.6667, A 0.000, B 0.000, C 0.000 }
gfCNCPoint3[17861] = {X 171.4215, Y 9.6405, Z -4.6667, A 0.000, B 0.000, C 0.000 }
gfCNCPoint3[17862] = {X 172.0576, Y 9.2779, Z -4.6667, A 0.000, B 0.000, C 0.000 }
gfCNCPoint3[17863] = {X 172.9936, Y 8.8768, Z -4.6667, A 0.000, B 0.000, C 0.000 }
gfCNCPoint3[17864] = {X 173.9926, Y 8.6787, Z -4.6667, A 0.000, B 0.000, C 0.000 }
gfCNCPoint3[17865] = {X 175.0109, Y 8.6923, Z -4.6667, A 0.000, B 0.000, C 0.000 }
gfCNCPoint3[17866] = {X 176.0042, Y 8.9169, Z -4.6667, A 0.000, B 0.000, C 0.000 }
gfCNCPoint3[17867] = {X 177.7753, Y 8.1692, Z -4.6667, A 0.000, B 0.000, C 0.000 }
gfCNCPoint3[17868] = {X 179.6001, Y 7.5639, Z -4.6667, A 0.000, B 0.000, C 0.000 }
gfCNCPoint3[17869] = {X 181.4670, Y 7.1050, Z -4.6667, A 0.000, B 0.000, C 0.000 }
gfCNCPoint3[17870] = {X 168.0206, Y 7.1050, Z -4.6667, A 0.000, B 0.000, C 0.000 }
gfCNCPoint3[17871] = {X 168.0206, Y 4.7050, Z -4.6667, A 0.000, B 0.000, C 0.000 }
gfCNCPoint3[17872] = {X 155.1591, Y 4.7050, Z -4.6667, A 0.000, B 0.000, C 0.000 }
gfCNCPoint3[17873] = {X 155.1591, Y 7.1050, Z -4.6667, A 0.000, B 0.000, C 0.000 }
gfCNCPoint3[17874] = {X 137.3637, Y 7.1050, Z -4.6667, A 0.000, B 0.000, C 0.000 }
gfCNCPoint3[17875] = {X 137.5335, Y 7.2914, Z -4.6667, A 0.000, B 0.000, C 0.000 }
gfCNCPoint3[17876] = {X 137.6935, Y 7.4864, Z -4.6667, A 0.000, B 0.000, C 0.000 }
gfCNCPoint3[17877] = {X 154.8293, Y 7.4864, Z -4.6667, A 0.000, B 0.000, C 0.000 }
gfCNCPoint3[17878] = {X 154.9892, Y 7.2914, Z -4.6667, A 0.000, B 0.000, C 0.000 }
gfCNCPoint3[17879] = {X 155.1591, Y 7.1050, Z -4.6667, A 0.000, B 0.000, C 0.000 }
gfCNCPoint3[17880] = {X 155.1591, Y 4.7050, Z -4.6667, A 0.000, B 0.000, C 0.000 }
gfCNCPoint3[17881] = {X 23.8352, Y 4.7050, Z -4.6667, A 0.000, B 0.000, C 0.000 }
gfCNCPoint3[17882] = {X 25.7636, Y 5.7850, Z -4.6667, A 0.000, B 0.000, C 0.000 }
gfCNCPoint3[17883] = {X 27.5758, Y 7.0504, Z -4.6667, A 0.000, B 0.000, C 0.000 }
gfCNCPoint3[17884] = {X 28.5590, Y 7.8748, Z -4.6667, A 0.000, B 0.000, C 0.000 }
gfCNCPoint3[17885] = {X 29.4805, Y 8.7676, Z -4.6667, A 0.000, B 0.000, C 0.000 }
gfCNCPoint3[17886] = {X 30.6888, Y 10.1629, Z -4.6667, A 0.000, B 0.000, C 0.000 }
gfCNCPoint3[17887] = {X 31.7468, Y 11.6753, Z -4.6667, A 0.000, B 0.000, C 0.000 }
gfCNCPoint3[17888] = {X 32.6431, Y 13.2888, Z -4.6667, A 0.000, B 0.000, C 0.000 }
gfCNCPoint3[17889] = {X 33.3684, Y 14.9860, Z -4.6667, A 0.000, B 0.000, C 0.000 }
gfCNCPoint3[17890] = {X 33.9188, Y 16.8170, Z -4.6667, A 0.000, B 0.000, C 0.000 }
gfCNCPoint3[17891] = {X 34.2906, Y 18.6924, Z -4.6667, A 0.000, B 0.000, C 0.000 }
gfCNCPoint3[17892] = {X 34.4805, Y 20.5949, Z -4.6667, A 0.000, B 0.000, C 0.000 }
gfCNCPoint3[17893] = {X 34.4867, Y 22.5068, Z -4.6667, A 0.000, B 0.000, C 0.000 }
gfCNCPoint3[17894] = {X 34.3091, Y 24.4104, Z -4.6667, A 0.000, B 0.000, C 0.000 }
gfCNCPoint3[17895] = {X 33.9493, Y 26.2882, Z -4.6667, A 0.000, B 0.000, C 0.000 }
gfCNCPoint3[17896] = {X 33.4656, Y 27.9397, Z -4.6667, A 0.000, B 0.000, C 0.000 }
gfCNCPoint3[17897] = {X 32.8132, Y 29.5321, Z -4.6667, A 0.000, B 0.000, C 0.000 }
gfCNCPoint3[17898] = {X 31.9992, Y 31.0483, Z -4.6667, A 0.000, B 0.000, C 0.000 }
gfCNCPoint3[17899] = {X 32.1287, Y 31.2841, Z -4.6667, A 0.000, B 0.000, C 0.000 }
gfCNCPoint3[17900] = {X 32.2512, Y 31.5235, Z -4.6667, A 0.000, B 0.000, C 0.000 }
gfCNCPoint3[17901] = {X 35.3025, Y 37.8269, Z -4.6667, A 0.000, B 0.000, C 0.000 }
gfCNCPoint3[17902] = {X 35.7263, Y 38.8573, Z -4.6667, A 0.000, B 0.000, C 0.000 }
gfCNCPoint3[17903] = {X 36.0224, Y 39.9313, Z -4.6667, A 0.000, B 0.000, C 0.000 }
gfCNCPoint3[17904] = {X 36.1865, Y 41.0332, Z -4.6667, A 0.000, B 0.000, C 0.000 }
gfCNCPoint3[17905] = {X 36.2163, Y 42.1469, Z -4.6667, A 0.000, B 0.000, C 0.000 }
gfCNCPoint3[17906] = {X 36.6304, Y 41.4262, Z -4.6667, A 0.000, B 0.000, C 0.000 }
gfCNCPoint3[17907] = {X 37.1608, Y 40.7862, Z -4.6667, A 0.000, B 0.000, C 0.000 }
gfCNCPoint3[17908] = {X 37.7922, Y 40.2454, Z -4.6667, A 0.000, B 0.000, C 0.000 }
gfCNCPoint3[17909] = {X 38.5061, Y 39.8197, Z -4.6667, A 0.000, B 0.000, C 0.000 }
gfCNCPoint3[17910] = {X 39.0448, Y 38.5340, Z -4.6667, A 0.000, B 0.000, C 0.000 }
gfCNCPoint3[17911] = {X 39.5406, Y 37.2311, Z -4.6667, A 0.000, B 0.000, C 0.000 }
gfCNCPoint3[17912] = {X 47.6703, Y 15.4045, Z -4.6667, A 0.000, B 0.000, C 0.000 }
gfCNCPoint3[17913] = {X 47.3200, Y 14.6512, Z -4.6667, A 0.000, B 0.000, C 0.000 }
gfCNCPoint3[17914] = {X 47.1026, Y 13.8493, Z -4.6667, A 0.000, B 0.000, C 0.000 }
gfCNCPoint3[17915] = {X 47.0244, Y 13.0222, Z -4.6667, A 0.000, B 0.000, C 0.000 }
gfCNCPoint3[17916] = {X 47.0242, Y 12.1868, Z -4.6667, A 0.000, B 0.000, C 0.000 }
gfCNCPoint3[17917] = {X 47.0722, Y 11.5041, Z -4.6667, A 0.000, B 0.000, C 0.000 }
gfCNCPoint3[17918] = {X 47.2153, Y 10.8348, Z -4.6667, A 0.000, B 0.000, C 0.000 }
gfCNCPoint3[17919] = {X 42.6031, Y 9.5050, Z -4.6667, A 0.000, B 0.000, C 0.000 }
gfCNCPoint3[17920] = {X 36.0457, Y 9.5050, Z -4.6667, A 0.000, B 0.000, C 0.000 }
gfCNCPoint3[17921] = {X 37.0556, Y 11.3879, Z -4.6667, A 0.000, B 0.000, C 0.000 }
gfCNCPoint3[17922] = {X 37.8838, Y 13.3575, Z -4.6667, A 0.000, B 0.000, C 0.000 }
gfCNCPoint3[17923] = {X 38.5468, Y 15.5388, Z -4.6667, A 0.000, B 0.000, C 0.000 }
gfCNCPoint3[17924] = {X 39.0056, Y 17.7719, Z -4.6667, A 0.000, B 0.000, C 0.000 }
gfCNCPoint3[17925] = {X 39.2563, Y 20.0378, Z -4.6667, A 0.000, B 0.000, C 0.000 }
gfCNCPoint3[17926] = {X 39.2967, Y 22.3172, Z -4.6667, A 0.000, B 0.000, C 0.000 }
gfCNCPoint3[17927] = {X 39.1266, Y 24.5906, Z -4.6667, A 0.000, B 0.000, C 0.000 }
gfCNCPoint3[17928] = {X 42.5394, Y 15.4280, Z -4.6667, A 0.000, B 0.000, C 0.000 }
gfCNCPoint3[17929] = {X 42.3075, Y 14.2452, Z -4.6667, A 0.000, B 0.000, C 0.000 }
gfCNCPoint3[17930] = {X 42.2244, Y 13.0428, Z -4.6667, A 0.000, B 0.000, C 0.000 }
gfCNCPoint3[17931] = {X 42.2242, Y 12.1868, Z -4.6667, A 0.000, B 0.000, C 0.000 }
gfCNCPoint3[17932] = {X 42.3194, Y 10.8326, Z -4.6667, A 0.000, B 0.000, C 0.000 }
gfCNCPoint3[17933] = {X 42.6031, Y 9.5050, Z -4.6667, A 0.000, B 0.000, C 0.000 }
gfCNCPoint3[17934] = {X 44.9092, Y 10.1699, Z -4.6667, A 0.000, B 0.000, C 0.000 }
gfCNCPoint3[17935] = {X 45.3323, Y 9.0550, Z -4.6667, A 0.000, B 0.000, C 0.000 }
gfCNCPoint3[17936] = {X 45.9317, Y 8.0241, Z -4.6667, A 0.000, B 0.000, C 0.000 }
gfCNCPoint3[17937] = {X 46.6914, Y 7.1050, Z -4.6667, A 0.000, B 0.000, C 0.000 }
gfCNCPoint3[17938] = {X 31.2113, Y 7.1050, Z -4.6667, A 0.000, B 0.000, C 0.000 }
gfCNCPoint3[17939] = {X 32.2268, Y 8.2450, Z -4.6667, A 0.000, B 0.000, C 0.000 }
gfCNCPoint3[17940] = {X 33.1536, Y 9.4582, Z -4.6667, A 0.000, B 0.000, C 0.000 }
gfCNCPoint3[17941] = {X 33.9865, Y 10.7377, Z -4.6667, A 0.000, B 0.000, C 0.000 }
gfCNCPoint3[17942] = {X 34.8870, Y 12.4162, Z -4.6667, A 0.000, B 0.000, C 0.000 }
gfCNCPoint3[17943] = {X 35.6261, Y 14.1718, Z -4.6667, A 0.000, B 0.000, C 0.000 }
gfCNCPoint3[17944] = {X 36.2230, Y 16.1388, Z -4.6667, A 0.000, B 0.000, C 0.000 }
gfCNCPoint3[17945] = {X 36.6359, Y 18.1526, Z -4.6667, A 0.000, B 0.000, C 0.000 }
gfCNCPoint3[17946] = {X 36.8615, Y 20.1959, Z -4.6667, A 0.000, B 0.000, C 0.000 }
gfCNCPoint3[17947] = {X 36.8976, Y 22.2512, Z -4.6667, A 0.000, B 0.000, C 0.000 }
gfCNCPoint3[17948] = {X 36.7441, Y 24.3011, Z -4.6667, A 0.000, B 0.000, C 0.000 }
gfCNCPoint3[17949] = {X 36.5507, Y 25.5810, Z -4.6667, A 0.000, B 0.000, C 0.000 }
gfCNCPoint3[17950] = {X 36.2833, Y 26.8475, Z -4.6667, A 0.000, B 0.000, C 0.000 }
gfCNCPoint3[17951] = {X 35.8744, Y 28.3067, Z -4.6667, A 0.000, B 0.000, C 0.000 }
gfCNCPoint3[17952] = {X 35.3504, Y 29.7285, Z -4.6667, A 0.000, B 0.000, C 0.000 }
gfCNCPoint3[17953] = {X 34.7145, Y 31.1040, Z -4.6667, A 0.000, B 0.000, C 0.000 }
gfCNCPoint3[17954] = {X 37.2844, Y 36.4128, Z -4.6667, A 0.000, B 0.000, C 0.000 }
gfCNCPoint3[17955] = {X 41.3757, Y 25.4283, Z -4.6667, A 0.000, B 0.000, C 0.000 }
gfCNCPoint3[17956] = {X 45.0743, Y 15.4981, Z -4.6667, A 0.000, B 0.000, C 0.000 }
gfCNCPoint3[17957] = {X 44.7425, Y 14.2853, Z -4.6667, A 0.000, B 0.000, C 0.000 }
gfCNCPoint3[17958] = {X 44.6244, Y 13.0334, Z -4.6667, A 0.000, B 0.000, C 0.000 }
gfCNCPoint3[17959] = {X 44.6242, Y 12.1868, Z -4.6667, A 0.000, B 0.000, C 0.000 }
gfCNCPoint3[17960] = {X 44.6958, Y 11.1683, Z -4.6667, A 0.000, B 0.000, C 0.000 }
gfCNCPoint3[17961] = {X 44.9092, Y 10.1699, Z -4.6667, A 0.000, B 0.000, C 0.000 }
gfCNCPoint3[17962] = {X 47.2153, Y 10.8348, Z -4.6667, A 0.000, B 0.000, C 0.000 }
gfCNCPoint3[17963] = {X 47.4989, Y 10.0875, Z -4.6667, A 0.000, B 0.000, C 0.000 }
gfCNCPoint3[17964] = {X 47.9007, Y 9.3965, Z -4.6667, A 0.000, B 0.000, C 0.000 }
gfCNCPoint3[17965] = {X 48.4099, Y 8.7803, Z -4.6667, A 0.000, B 0.000, C 0.000 }
gfCNCPoint3[17966] = {X 49.1545, Y 8.1553, Z -4.6667, A 0.000, B 0.000, C 0.000 }
gfCNCPoint3[17967] = {X 50.0081, Y 7.6903, Z -4.6667, A 0.000, B 0.000, C 0.000 }
gfCNCPoint3[17968] = {X 50.9370, Y 7.4036, Z -4.6667, A 0.000, B 0.000, C 0.000 }
gfCNCPoint3[17969] = {X 51.9042, Y 7.3068, Z -4.6667, A 0.000, B 0.000, C 0.000 }
gfCNCPoint3[17970] = {X 59.6221, Y 7.3068, Z -4.6667, A 0.000, B 0.000, C 0.000 }
gfCNCPoint3[17971] = {X 60.5894, Y 7.4036, Z -4.6667, A 0.000, B 0.000, C 0.000 }
gfCNCPoint3[17972] = {X 61.5183, Y 7.6903, Z -4.6667, A 0.000, B 0.000, C 0.000 }
gfCNCPoint3[17973] = {X 62.3719, Y 8.1553, Z -4.6667, A 0.000, B 0.000, C 0.000 }
gfCNCPoint3[17974] = {X 63.1164, Y 8.7803, Z -4.6667, A 0.000, B 0.000, C 0.000 }
gfCNCPoint3[17975] = {X 63.7054, Y 9.5145, Z -4.6667, A 0.000, B 0.000, C 0.000 }
gfCNCPoint3[17976] = {X 64.1424, Y 10.3480, Z -4.6667, A 0.000, B 0.000, C 0.000 }
gfCNCPoint3[17977] = {X 64.4114, Y 11.2500, Z -4.6667, A 0.000, B 0.000, C 0.000 }
gfCNCPoint3[17978] = {X 64.5021, Y 12.1868, Z -4.6667, A 0.000, B 0.000, C 0.000 }
gfCNCPoint3[17979] = {X 64.5019, Y 13.0237, Z -4.6667, A 0.000, B 0.000, C 0.000 }
gfCNCPoint3[17980] = {X 64.4204, Y 13.8674, Z -4.6667, A 0.000, B 0.000, C 0.000 }
gfCNCPoint3[17981] = {X 64.1941, Y 14.6842, Z -4.6667, A 0.000, B 0.000, C 0.000 }
gfCNCPoint3[17982] = {X 63.8300, Y 15.4496, Z -4.6667, A 0.000, B 0.000, C 0.000 }
gfCNCPoint3[17983] = {X 72.9544, Y 39.8579, Z -4.6667, A 0.000, B 0.000, C 0.000 }
gfCNCPoint3[17984] = {X 73.8444, Y 40.4399, Z -4.6667, A 0.000, B 0.000, C 0.000 }
gfCNCPoint3[17985] = {X 74.5871, Y 41.2008, Z -4.6667, A 0.000, B 0.000, C 0.000 }
gfCNCPoint3[17986] = {X 75.1475, Y 42.1045, Z -4.6667, A 0.000, B 0.000, C 0.000 }
gfCNCPoint3[17987] = {X 75.4987, Y 43.1081, Z -4.6667, A 0.000, B 0.000, C 0.000 }
gfCNCPoint3[17988] = {X 75.6243, Y 44.1640, Z -4.6667, A 0.000, B 0.000, C 0.000 }
gfCNCPoint3[17989] = {X 75.6245, Y 45.0000, Z -4.6667, A 0.000, B 0.000, C 0.000 }
gfCNCPoint3[17990] = {X 75.5307, Y 45.9520, Z -4.6667, A 0.000, B 0.000, C 0.000 }
gfCNCPoint3[17991] = {X 75.2530, Y 46.8675, Z -4.6667, A 0.000, B 0.000, C 0.000 }
gfCNCPoint3[17992] = {X 74.8020, Y 47.7112, Z -4.6667, A 0.000, B 0.000, C 0.000 }
gfCNCPoint3[17993] = {X 74.1951, Y 48.4507, Z -4.6667, A 0.000, B 0.000, C 0.000 }
gfCNCPoint3[17994] = {X 73.4556, Y 49.0576, Z -4.6667, A 0.000, B 0.000, C 0.000 }
gfCNCPoint3[17995] = {X 72.6120, Y 49.5085, Z -4.6667, A 0.000, B 0.000, C 0.000 }
gfCNCPoint3[17996] = {X 71.6965, Y 49.7862, Z -4.6667, A 0.000, B 0.000, C 0.000 }
gfCNCPoint3[17997] = {X 70.7445, Y 49.8800, Z -4.6667, A 0.000, B 0.000, C 0.000 }
gfCNCPoint3[17998] = {X 64.1851, Y 49.8800, Z -4.6667, A 0.000, B 0.000, C 0.000 }
gfCNCPoint3[17999] = {X 63.2331, Y 49.7862, Z -4.6667, A 0.000, B 0.000, C 0.000 }
gfCNCPoint3[18000] = {X 62.3176, Y 49.5085, Z -4.6667, A 0.000, B 0.000, C 0.000 }
gfCNCPoint3[18001] = {X 61.4740, Y 49.0576, Z -4.6667, A 0.000, B 0.000, C 0.000 }
gfCNCPoint3[18002] = {X 60.7345, Y 48.4507, Z -4.6667, A 0.000, B 0.000, C 0.000 }
gfCNCPoint3[18003] = {X 60.1276, Y 47.7112, Z -4.6667, A 0.000, B 0.000, C 0.000 }
gfCNCPoint3[18004] = {X 59.6766, Y 46.8675, Z -4.6667, A 0.000, B 0.000, C 0.000 }
gfCNCPoint3[18005] = {X 59.3989, Y 45.9520, Z -4.6667, A 0.000, B 0.000, C 0.000 }
gfCNCPoint3[18006] = {X 59.3051, Y 45.0000, Z -4.6667, A 0.000, B 0.000, C 0.000 }
gfCNCPoint3[18007] = {X 59.3052, Y 44.2029, Z -4.6667, A 0.000, B 0.000, C 0.000 }
gfCNCPoint3[18008] = {X 59.3847, Y 43.3311, Z -4.6667, A 0.000, B 0.000, C 0.000 }
gfCNCPoint3[18009] = {X 59.6188, Y 42.4876, Z -4.6667, A 0.000, B 0.000, C 0.000 }
gfCNCPoint3[18010] = {X 59.9997, Y 41.6994, Z -4.6667, A 0.000, B 0.000, C 0.000 }
gfCNCPoint3[18011] = {X 59.6155, Y 40.6492, Z -4.6667, A 0.000, B 0.000, C 0.000 }
gfCNCPoint3[18012] = {X 52.4664, Y 40.6492, Z -4.6667, A 0.000, B 0.000, C 0.000 }
gfCNCPoint3[18013] = {X 51.9469, Y 42.0449, Z -4.6667, A 0.000, B 0.000, C 0.000 }
gfCNCPoint3[18014] = {X 52.2216, Y 42.7242, Z -4.6667, A 0.000, B 0.000, C 0.000 }
gfCNCPoint3[18015] = {X 52.3915, Y 43.4370, Z -4.6667, A 0.000, B 0.000, C 0.000 }
gfCNCPoint3[18016] = {X 52.4528, Y 44.1672, Z -4.6667, A 0.000, B 0.000, C 0.000 }
gfCNCPoint3[18017] = {X 52.4529, Y 45.0000, Z -4.6667, A 0.000, B 0.000, C 0.000 }
gfCNCPoint3[18018] = {X 52.3592, Y 45.9520, Z -4.6667, A 0.000, B 0.000, C 0.000 }
gfCNCPoint3[18019] = {X 52.0815, Y 46.8675, Z -4.6667, A 0.000, B 0.000, C 0.000 }
gfCNCPoint3[18020] = {X 51.6305, Y 47.7112, Z -4.6667, A 0.000, B 0.000, C 0.000 }
gfCNCPoint3[18021] = {X 51.0236, Y 48.4507, Z -4.6667, A 0.000, B 0.000, C 0.000 }
gfCNCPoint3[18022] = {X 50.2841, Y 49.0576, Z -4.6667, A 0.000, B 0.000, C 0.000 }
gfCNCPoint3[18023] = {X 49.4404, Y 49.5085, Z -4.6667, A 0.000, B 0.000, C 0.000 }
gfCNCPoint3[18024] = {X 48.5250, Y 49.7862, Z -4.6667, A 0.000, B 0.000, C 0.000 }
gfCNCPoint3[18025] = {X 47.5729, Y 49.8800, Z -4.6667, A 0.000, B 0.000, C 0.000 }
gfCNCPoint3[18026] = {X 40.6393, Y 49.8800, Z -4.6667, A 0.000, B 0.000, C 0.000 }
gfCNCPoint3[18027] = {X 39.6433, Y 49.7773, Z -4.6667, A 0.000, B 0.000, C 0.000 }
gfCNCPoint3[18028] = {X 38.6892, Y 49.4734, Z -4.6667, A 0.000, B 0.000, C 0.000 }
gfCNCPoint3[18029] = {X 37.8173, Y 48.9813, Z -4.6667, A 0.000, B 0.000, C 0.000 }
gfCNCPoint3[18030] = {X 37.0641, Y 48.3215, Z -4.6667, A 0.000, B 0.000, C 0.000 }
gfCNCPoint3[18031] = {X 36.5085, Y 47.5983, Z -4.6667, A 0.000, B 0.000, C 0.000 }
gfCNCPoint3[18032] = {X 36.0972, Y 46.7843, Z -4.6667, A 0.000, B 0.000, C 0.000 }
